C03596=1036.829,292.266,-117.984,171.449,43.308,158.322
C03597=1036.819,291.919,-117.939,171.445,43.306,158.321
C03598=1036.810,291.572,-117.895,171.438,43.304,158.320
C03599=1036.801,291.226,-117.849,171.434,43.302,158.319
C03600=1036.791,290.879,-117.804,171.429,43.301,158.318
C03601=1036.784,290.631,-117.772,171.425,43.299,158.318
C03602=1036.777,290.384,-117.740,171.420,43.298,158.317
C03603=1036.771,290.136,-117.708,171.417,43.297,158.317
C03604=1036.763,289.888,-117.676,171.413,43.296,158.316
C03605=1036.757,289.640,-117.644,171.409,43.295,158.316
C03606=1036.750,289.393,-117.612,171.406,43.294,158.315
C03607=1036.744,289.144,-117.580,171.402,43.292,158.314
C03608=1036.737,288.896,-117.549,171.398,43.291,158.314
C03609=1036.729,288.648,-117.516,171.395,43.290,158.313
C03610=1036.723,288.401,-117.485,171.391,43.288,158.313
C03611=1036.716,288.153,-117.453,171.386,43.287,158.312
C03612=1036.710,287.905,-117.420,171.383,43.286,158.311
C03613=1036.703,287.657,-117.389,171.379,43.285,158.311
C03614=1036.696,287.410,-117.357,171.375,43.284,158.310
C03615=1036.689,287.162,-117.325,171.372,43.283,158.310
C03616=1036.682,286.913,-117.294,171.368,43.281,158.309
C03617=1036.675,286.666,-117.261,171.364,43.280,158.309
C03618=1036.669,286.418,-117.230,171.361,43.279,158.308
C03619=1036.662,286.170,-117.198,171.357,43.278,158.308
C03620=1036.655,285.922,-117.167,171.354,43.277,158.307
C03621=1036.648,285.675,-117.134,171.350,43.276,158.307
C03622=1036.642,285.427,-117.103,171.346,43.275,158.306
C03623=1036.634,285.178,-117.071,171.343,43.274,158.306
C03624=1036.627,284.930,-117.040,171.339,43.272,158.305
C03625=1036.621,284.683,-117.008,171.336,43.272,158.305
C03626=1036.613,284.435,-116.978,171.331,43.270,158.304
C03627=1036.607,284.187,-116.946,171.327,43.269,158.303
C03628=1036.600,283.940,-116.914,171.323,43.268,158.303
C03629=1036.593,283.692,-116.883,171.320,43.267,158.302
C03630=1036.586,283.444,-116.851,171.316,43.266,158.302
C03631=1036.579,283.196,-116.820,171.313,43.265,158.301
C03632=1036.573,282.948,-116.788,171.309,43.264,158.301
C03633=1036.566,282.700,-116.757,171.305,43.263,158.300
C03634=1036.559,282.452,-116.725,171.302,43.261,158.300
C03635=1036.552,282.204,-116.694,171.298,43.261,158.299
C03636=1036.546,281.957,-116.663,171.295,43.259,158.299
C03637=1036.539,281.709,-116.631,171.291,43.258,158.298
C03638=1036.532,281.461,-116.600,171.287,43.257,158.298
C03639=1036.526,281.213,-116.568,171.284,43.256,158.297
C03640=1036.519,280.965,-116.537,171.280,43.255,158.297
C03641=1036.512,280.717,-116.505,171.277,43.254,158.296
C03642=1036.506,280.468,-116.475,171.273,43.253,158.295
C03643=1036.499,280.221,-116.443,171.270,43.252,158.295
C03644=1036.492,279.973,-116.412,171.266,43.251,158.294
C03645=1036.485,279.725,-116.380,171.262,43.250,158.294
C03646=1036.479,279.477,-116.349,171.259,43.249,158.293
C03647=1036.472,279.229,-116.317,171.255,43.247,158.293
C03648=1036.465,278.981,-116.286,171.252,43.247,158.292
C03649=1036.459,278.733,-116.255,171.249,43.245,158.292
C03650=1036.452,278.485,-116.224,171.245,43.244,158.291
C03651=1036.445,278.237,-116.193,171.242,43.243,158.291
C03652=1036.438,277.989,-116.162,171.238,43.242,158.290
C03653=1036.429,277.655,-116.119,171.233,43.241,158.290
C03654=1036.420,277.319,-116.078,171.229,43.240,158.289
C03655=1036.411,276.985,-116.036,171.224,43.238,158.288
C03656=1036.401,276.651,-115.994,171.219,43.237,158.288
C03657=1036.395,276.402,-115.964,171.216,43.236,158.287
C03658=1036.388,276.154,-115.932,171.212,43.235,158.287
C03659=1036.382,275.906,-115.902,171.208,43.234,158.286
C03660=1036.374,275.658,-115.871,171.205,43.233,158.286
C03661=1036.368,275.411,-115.840,171.201,43.232,158.285
C03662=1036.362,275.162,-115.809,171.198,43.231,158.285
C03663=1036.354,274.915,-115.778,171.194,43.230,158.284
C03664=1036.348,274.666,-115.747,171.191,43.229,158.284
C03665=1036.341,274.418,-115.716,171.187,43.228,158.283
C03666=1036.335,274.170,-115.685,171.185,43.227,158.283
C03667=1036.328,273.923,-115.655,171.181,43.226,158.282
C03668=1036.321,273.674,-115.624,171.177,43.225,158.282
C03669=1036.314,273.427,-115.593,171.174,43.224,158.281
C03670=1036.308,273.178,-115.562,171.170,43.223,158.281
C03671=1036.301,272.930,-115.531,171.167,43.222,158.280
C03672=1036.294,272.682,-115.501,171.163,43.222,158.280
C03673=1036.288,272.434,-115.471,171.160,43.220,158.279
C03674=1036.280,272.187,-115.440,171.156,43.220,158.279
C03675=1036.274,271.938,-115.409,171.153,43.219,158.279
C03676=1036.267,271.690,-115.378,171.150,43.217,158.278
C03677=1036.260,271.442,-115.347,171.147,43.217,158.278
C03678=1036.254,271.194,-115.317,171.143,43.216,158.277
C03679=1036.247,270.947,-115.286,171.139,43.215,158.277
C03680=1036.240,270.698,-115.256,171.136,43.214,158.276
C03681=1036.233,270.450,-115.225,171.132,43.213,158.276
C03682=1036.227,270.202,-115.195,171.129,43.212,158.275
C03683=1036.220,269.955,-115.164,171.126,43.211,158.275
C03684=1036.214,269.706,-115.134,171.123,43.210,158.274
C03685=1036.206,269.458,-115.103,171.119,43.210,158.274
C03686=1036.201,269.210,-115.073,171.116,43.208,158.273
C03687=1036.193,268.962,-115.042,171.112,43.208,158.273
C03688=1036.187,268.714,-115.011,171.109,43.207,158.272
C03689=1036.180,268.466,-114.981,171.105,43.206,158.272
C03690=1036.173,268.218,-114.952,171.103,43.205,158.272
C03691=1036.167,267.970,-114.921,171.099,43.204,158.271
C03692=1036.159,267.721,-114.891,171.096,43.203,158.271
C03693=1036.154,267.474,-114.860,171.092,43.203,158.270
C03694=1036.146,267.225,-114.830,171.089,43.202,158.270
C03695=1036.140,266.977,-114.799,171.085,43.201,158.269
C03696=1036.133,266.730,-114.769,171.083,43.200,158.269
C03697=1036.126,266.482,-114.739,171.079,43.199,158.268
C03698=1036.120,266.233,-114.708,171.076,43.198,158.268
C03699=1036.113,265.986,-114.679,171.072,43.198,158.268
C03700=1036.106,265.737,-114.648,171.069,43.197,158.267
C03701=1036.099,265.489,-114.618,171.066,43.195,158.267
C03702=1036.093,265.241,-114.588,171.063,43.195,158.266
C03703=1036.086,264.993,-114.559,171.059,43.194,158.266
C03704=1036.079,264.744,-114.528,171.056,43.193,158.265
C03705=1036.073,264.497,-114.498,171.052,43.193,158.265
C03706=1036.066,264.248,-114.468,171.050,43.192,158.265
C03707=1036.059,264.000,-114.438,171.046,43.191,158.264
C03708=1036.052,263.753,-114.408,171.043,43.190,158.264
C03709=1036.044,263.422,-114.368,171.038,43.189,158.263
C03710=1036.035,263.092,-114.328,171.035,43.188,158.263
C03711=1036.026,262.762,-114.287,171.030,43.187,158.262
C03712=1036.017,262.432,-114.248,171.025,43.185,158.261
C03713=1036.009,262.184,-114.218,171.022,43.185,158.261
C03714=1036.004,261.935,-114.188,171.019,43.184,158.260
C03715=1035.997,261.687,-114.158,171.016,43.183,158.260
C03716=1035.990,261.440,-114.128,171.012,43.182,158.260
C03717=1035.983,261.192,-114.098,171.009,43.182,158.259
C03718=1035.976,260.943,-114.069,171.006,43.181,158.259
C03719=1035.970,260.695,-114.039,171.003,43.180,158.258
C03720=1035.963,260.446,-114.009,171.000,43.179,158.258
C03721=1035.956,260.199,-113.980,170.996,43.179,158.258
C03722=1035.948,259.951,-113.950,170.993,43.179,158.257
C03723=1035.942,259.702,-113.921,170.990,43.178,158.257
C03724=1035.935,259.455,-113.891,170.987,43.177,158.256
C03725=1035.928,259.206,-113.862,170.983,43.176,158.256
C03726=1035.922,258.958,-113.832,170.980,43.176,158.256
C03727=1035.915,258.709,-113.802,170.978,43.175,158.255
C03728=1035.908,258.462,-113.773,170.974,43.174,158.255
C03729=1035.901,258.214,-113.743,170.971,43.173,158.254
C03730=1035.894,257.965,-113.713,170.967,43.173,158.254
C03731=1035.887,257.718,-113.684,170.965,43.172,158.254
C03732=1035.880,257.469,-113.655,170.961,43.172,158.253
C03733=1035.874,257.221,-113.626,170.958,43.171,158.253
C03734=1035.867,256.972,-113.595,170.955,43.170,158.252
C03735=1035.860,256.724,-113.566,170.952,43.169,158.252
C03736=1035.853,256.476,-113.536,170.949,43.169,158.252
C03737=1035.847,256.228,-113.507,170.945,43.168,158.251
C03738=1035.840,255.980,-113.477,170.943,43.167,158.251
C03739=1035.833,255.732,-113.449,170.939,43.167,158.251
C03740=1035.826,255.483,-113.419,170.936,43.166,158.250
C03741=1035.819,255.236,-113.389,170.933,43.165,158.250
C03742=1035.813,254.987,-113.360,170.930,43.165,158.249
C03743=1035.806,254.739,-113.330,170.927,43.164,158.249
C03744=1035.800,254.491,-113.301,170.923,43.163,158.248
C03745=1035.793,254.242,-113.272,170.921,43.162,158.248
C03746=1035.786,253.995,-113.243,170.917,43.162,158.248
C03747=1035.779,253.746,-113.213,170.914,43.161,158.247
C03748=1035.772,253.498,-113.184,170.912,43.161,158.247
C03749=1035.765,253.250,-113.154,170.908,43.160,158.247
C03750=1035.759,253.002,-113.125,170.905,43.159,158.246
C03751=1035.753,252.754,-113.096,170.902,43.158,158.246
C03752=1035.746,252.505,-113.067,170.899,43.158,158.245
C03753=1035.739,252.258,-113.037,170.895,43.157,158.245
C03754=1035.732,252.009,-113.008,170.893,43.157,158.245
C03755=1035.726,251.761,-112.979,170.890,43.156,158.244
C03756=1035.719,251.513,-112.950,170.886,43.155,158.244
C03757=1035.712,251.264,-112.921,170.884,43.154,158.244
C03758=1035.706,251.016,-112.891,170.880,43.154,158.243
C03759=1035.700,250.768,-112.862,170.877,43.153,158.243
C03760=1035.692,250.520,-112.833,170.874,43.153,158.242
C03761=1035.686,250.271,-112.804,170.871,43.152,158.242
C03762=1035.680,250.023,-112.775,170.869,43.151,158.242
C03763=1035.673,249.774,-112.745,170.865,43.150,158.241
C03764=1035.666,249.527,-112.716,170.862,43.149,158.241
C03765=1035.657,249.195,-112.677,170.858,43.149,158.240
C03766=1035.648,248.864,-112.638,170.854,43.148,158.240
C03767=1035.640,248.532,-112.600,170.850,43.147,158.239
C03768=1035.631,248.201,-112.560,170.846,43.146,158.239
C03769=1035.625,247.953,-112.531,170.843,43.145,158.238
C03770=1035.618,247.705,-112.502,170.840,43.145,158.238
C03771=1035.611,247.456,-112.473,170.837,43.144,158.238
C03772=1035.604,247.208,-112.444,170.834,43.144,158.237
C03773=1035.598,246.960,-112.415,170.831,43.143,158.237
C03774=1035.592,246.712,-112.386,170.828,43.142,158.237
C03775=1035.585,246.463,-112.357,170.825,43.141,158.236
C03776=1035.579,246.215,-112.328,170.822,43.140,158.236
C03777=1035.572,245.967,-112.299,170.819,43.140,158.236
C03778=1035.566,245.719,-112.270,170.816,43.139,158.235
C03779=1035.559,245.470,-112.241,170.813,43.139,158.235
C03780=1035.553,245.222,-112.212,170.811,43.138,158.234
C03781=1035.546,244.974,-112.183,170.807,43.137,158.234
C03782=1035.539,244.726,-112.154,170.805,43.137,158.234
C03783=1035.533,244.477,-112.126,170.801,43.136,158.233
C03784=1035.527,244.228,-112.097,170.798,43.135,158.233
C03785=1035.520,243.980,-112.068,170.796,43.135,158.233
C03786=1035.513,243.732,-112.039,170.792,43.134,158.232
C03787=1035.506,243.484,-112.011,170.790,43.134,158.232
C03788=1035.500,243.235,-111.982,170.786,43.133,158.232
C03789=1035.493,242.987,-111.954,170.784,43.133,158.231
C03790=1035.487,242.739,-111.925,170.781,43.132,158.231
C03791=1035.480,242.491,-111.896,170.778,43.132,158.230
C03792=1035.474,242.243,-111.868,170.775,43.131,158.230
C03793=1035.467,241.994,-111.838,170.771,43.130,158.230
C03794=1035.460,241.746,-111.810,170.769,43.130,158.229
C03795=1035.453,241.498,-111.781,170.766,43.129,158.229
C03796=1035.447,241.249,-111.753,170.763,43.128,158.229
C03797=1035.441,241.001,-111.724,170.760,43.128,158.228
C03798=1035.434,240.753,-111.696,170.758,43.127,158.228
C03799=1035.428,240.505,-111.667,170.754,43.126,158.228
C03800=1035.420,240.256,-111.639,170.752,43.126,158.227
C03801=1035.413,240.008,-111.610,170.748,43.125,158.227
C03802=1035.407,239.759,-111.582,170.746,43.125,158.227
C03803=1035.400,239.512,-111.553,170.743,43.124,158.226
C03804=1035.393,239.263,-111.526,170.740,43.124,158.226
C03805=1035.387,239.014,-111.496,170.737,43.123,158.226
C03806=1035.380,238.766,-111.468,170.735,43.123,158.225
C03807=1035.373,238.518,-111.440,170.731,43.122,158.225
C03808=1035.366,238.270,-111.412,170.729,43.122,158.225
C03809=1035.360,238.022,-111.383,170.726,43.121,158.224
C03810=1035.353,237.773,-111.356,170.723,43.121,158.224
C03811=1035.346,237.525,-111.327,170.720,43.120,158.224
C03812=1035.340,237.277,-111.299,170.718,43.120,158.223
C03813=1035.333,237.028,-111.270,170.714,43.119,158.223
C03814=1035.326,236.780,-111.242,170.712,43.119,158.223
C03815=1035.319,236.531,-111.214,170.709,43.118,158.222
C03816=1035.312,236.283,-111.186,170.706,43.118,158.222
C03817=1035.306,236.035,-111.158,170.703,43.117,158.222
C03818=1035.300,235.787,-111.129,170.700,43.117,158.221
C03819=1035.293,235.538,-111.102,170.697,43.116,158.221
C03820=1035.286,235.290,-111.074,170.695,43.116,158.221
C03821=1035.277,234.952,-111.035,170.690,43.115,158.220
C03822=1035.269,234.615,-110.997,170.687,43.114,158.220
C03823=1035.259,234.278,-110.958,170.682,43.114,158.219
C03824=1035.250,233.940,-110.920,170.679,43.113,158.219
C03825=1035.243,233.691,-110.892,170.677,43.113,158.219
C03826=1035.236,233.444,-110.864,170.673,43.112,158.218
C03827=1035.230,233.195,-110.836,170.671,43.112,158.218
C03828=1035.223,232.947,-110.808,170.667,43.111,158.218
C03829=1035.217,232.698,-110.780,170.665,43.111,158.217
C03830=1035.210,232.450,-110.752,170.662,43.110,158.217
C03831=1035.203,232.202,-110.724,170.660,43.110,158.217
C03832=1035.197,231.953,-110.696,170.657,43.109,158.216
C03833=1035.191,231.704,-110.668,170.654,43.109,158.216
C03834=1035.184,231.457,-110.639,170.651,43.108,158.216
C03835=1035.177,231.208,-110.612,170.648,43.108,158.215
C03836=1035.170,230.960,-110.584,170.646,43.107,158.215
C03837=1035.164,230.711,-110.556,170.642,43.107,158.215
C03838=1035.157,230.463,-110.528,170.640,43.106,158.214
C03839=1035.150,230.214,-110.501,170.638,43.106,158.214
C03840=1035.144,229.966,-110.473,170.635,43.105,158.214
C03841=1035.137,229.718,-110.445,170.632,43.105,158.213
C03842=1035.130,229.470,-110.417,170.629,43.104,158.213
C03843=1035.123,229.221,-110.389,170.627,43.104,158.213
C03844=1035.117,228.974,-110.362,170.624,43.103,158.213
C03845=1035.110,228.725,-110.334,170.621,43.103,158.212
C03846=1035.104,228.477,-110.306,170.618,43.102,158.212
C03847=1035.097,228.228,-110.279,170.615,43.102,158.212
C03848=1035.090,227.980,-110.251,170.613,43.101,158.211
C03849=1035.084,227.731,-110.223,170.609,43.101,158.211
C03850=1035.077,227.483,-110.195,170.607,43.101,158.211
C03851=1035.070,227.234,-110.168,170.605,43.101,158.211
C03852=1035.064,226.986,-110.140,170.602,43.100,158.210
C03853=1035.057,226.738,-110.112,170.599,43.100,158.210
C03854=1035.050,226.489,-110.085,170.596,43.099,158.210
C03855=1035.043,226.241,-110.057,170.594,43.099,158.209
C03856=1035.037,225.992,-110.030,170.591,43.098,158.209
C03857=1035.030,225.743,-110.003,170.588,43.098,158.209
C03858=1035.023,225.495,-109.975,170.586,43.097,158.208
C03859=1035.017,225.247,-109.947,170.582,43.097,158.208
C03860=1035.009,224.998,-109.920,170.580,43.097,158.208
C03861=1035.003,224.751,-109.893,170.578,43.096,158.207
C03862=1034.996,224.502,-109.865,170.575,43.096,158.207
C03863=1034.990,224.253,-109.838,170.572,43.096,158.207
C03864=1034.983,224.005,-109.810,170.570,43.095,158.207
C03865=1034.977,223.756,-109.782,170.567,43.095,158.206
C03866=1034.969,223.508,-109.755,170.564,43.094,158.206
C03867=1034.963,223.260,-109.728,170.561,43.094,158.206
C03868=1034.956,223.011,-109.701,170.559,43.093,158.205
C03869=1034.950,222.763,-109.673,170.556,43.093,158.205
C03870=1034.943,222.515,-109.645,170.553,43.093,158.205
C03871=1034.936,222.266,-109.618,170.551,43.092,158.205
C03872=1034.930,222.017,-109.591,170.549,43.092,158.204
C03873=1034.923,221.769,-109.564,170.545,43.092,158.204
C03874=1034.916,221.520,-109.536,170.543,43.091,158.204
C03875=1034.910,221.273,-109.508,170.541,43.090,158.203
C03876=1034.903,221.024,-109.482,170.537,43.090,158.203
C03877=1034.894,220.679,-109.444,170.534,43.090,158.203
C03878=1034.885,220.334,-109.406,170.530,43.089,158.202
C03879=1034.875,219.989,-109.368,170.527,43.088,158.202
C03880=1034.866,219.644,-109.330,170.523,43.087,158.201
C03881=1034.860,219.395,-109.302,170.520,43.087,158.201
C03882=1034.853,219.148,-109.276,170.518,43.087,158.201
C03883=1034.846,218.899,-109.249,170.516,43.087,158.201
C03884=1034.839,218.651,-109.221,170.513,43.087,158.200
C03885=1034.833,218.402,-109.194,170.510,43.086,158.200
C03886=1034.825,218.154,-109.167,170.508,43.085,158.200
C03887=1034.819,217.905,-109.140,170.505,43.085,158.200
C03888=1034.812,217.657,-109.113,170.502,43.085,158.199
C03889=1034.806,217.408,-109.086,170.500,43.085,158.199
C03890=1034.798,217.160,-109.059,170.497,43.084,158.199
C03891=1034.792,216.911,-109.032,170.494,43.084,158.198
C03892=1034.786,216.663,-109.005,170.492,43.083,158.198
C03893=1034.779,216.414,-108.979,170.489,43.083,158.198
C03894=1034.772,216.166,-108.951,170.487,43.083,158.198
C03895=1034.765,215.917,-108.924,170.484,43.082,158.197
C03896=1034.759,215.669,-108.897,170.481,43.082,158.197
C03897=1034.752,215.421,-108.871,170.479,43.082,158.197
C03898=1034.745,215.172,-108.844,170.477,43.081,158.197
C03899=1034.738,214.924,-108.816,170.474,43.081,158.196
C03900=1034.732,214.675,-108.790,170.471,43.080,158.196
C03901=1034.725,214.427,-108.763,170.469,43.080,158.196
C03902=1034.718,214.178,-108.736,170.466,43.080,158.196
C03903=1034.711,213.929,-108.709,170.464,43.079,158.195
C03904=1034.705,213.681,-108.682,170.461,43.079,158.195
C03905=1034.698,213.433,-108.655,170.459,43.079,158.195
C03906=1034.692,213.184,-108.628,170.456,43.078,158.194
C03907=1034.685,212.936,-108.602,170.454,43.078,158.194
C03908=1034.678,212.687,-108.575,170.451,43.078,158.194
C03909=1034.671,212.438,-108.548,170.449,43.078,158.194
C03910=1034.665,212.191,-108.521,170.446,43.077,158.193
C03911=1034.658,211.942,-108.494,170.444,43.076,158.193
C03912=1034.652,211.693,-108.467,170.441,43.076,158.193
C03913=1034.645,211.445,-108.441,170.438,43.076,158.193
C03914=1034.639,211.196,-108.414,170.436,43.076,158.192
C03915=1034.631,210.948,-108.387,170.434,43.075,158.192
C03916=1034.625,210.700,-108.361,170.430,43.075,158.192
C03917=1034.618,210.451,-108.333,170.428,43.074,158.191
C03918=1034.611,210.202,-108.307,170.426,43.074,158.191
C03919=1034.605,209.954,-108.281,170.424,43.074,158.191
C03920=1034.598,209.705,-108.254,170.420,43.074,158.191
C03921=1034.591,209.457,-108.228,170.418,43.073,158.190
C03922=1034.585,209.208,-108.201,170.416,43.073,158.190
C03923=1034.578,208.960,-108.174,170.414,43.073,158.190
C03924=1034.571,208.712,-108.148,170.411,43.072,158.190
C03925=1034.564,208.463,-108.121,170.408,43.072,158.189
C03926=1034.558,208.214,-108.094,170.406,43.071,158.189
C03927=1034.551,207.966,-108.068,170.404,43.071,158.189
C03928=1034.544,207.717,-108.042,170.401,43.071,158.189
C03929=1034.537,207.469,-108.015,170.398,43.071,158.188
C03930=1034.531,207.220,-107.989,170.396,43.071,158.188
C03931=1034.524,206.972,-107.962,170.394,43.070,158.188
C03932=1034.518,206.723,-107.936,170.391,43.070,158.188
C03933=1034.508,206.384,-107.900,170.388,43.069,158.187
C03934=1034.498,206.045,-107.864,170.385,43.069,158.187
C03935=1034.490,205.706,-107.828,170.381,43.068,158.187
C03936=1034.481,205.366,-107.792,170.378,43.068,158.186
C03937=1034.454,204.316,-107.686,170.052,42.963,158.140
C03938=1034.448,204.068,-107.661,170.048,42.964,158.140
C03939=1034.443,203.820,-107.636,170.045,42.965,158.140
C03940=1034.436,203.571,-107.611,170.042,42.965,158.140
C03941=1034.430,203.322,-107.586,170.038,42.966,158.139
C03942=1034.424,203.073,-107.561,170.034,42.966,158.139
C03943=1034.417,202.825,-107.536,170.031,42.966,158.139
C03944=1034.412,202.577,-107.511,170.027,42.967,158.139
C03945=1034.406,202.327,-107.486,170.024,42.967,158.139
C03946=1034.400,202.079,-107.461,170.021,42.968,158.139
C03947=1034.393,201.830,-107.435,170.018,42.968,158.138
C03948=1034.388,201.581,-107.411,170.014,42.969,158.138
C03949=1034.381,201.333,-107.386,170.011,42.969,158.138
C03950=1034.375,201.084,-107.361,170.008,42.970,158.138
C03951=1034.369,200.835,-107.337,170.004,42.970,158.138
C03952=1034.363,200.587,-107.311,170.001,42.971,158.138
C03953=1034.357,200.337,-107.287,169.998,42.971,158.137
C03954=1034.351,200.090,-107.262,169.994,42.972,158.137
C03955=1034.345,199.840,-107.238,169.991,42.972,158.137
C03956=1034.338,199.592,-107.213,169.987,42.973,158.137
C03957=1034.332,199.343,-107.188,169.984,42.973,158.137
C03958=1034.325,199.094,-107.163,169.980,42.974,158.137
C03959=1034.320,198.846,-107.139,169.977,42.975,158.137
C03960=1034.313,198.597,-107.114,169.974,42.975,158.137
C03961=1034.307,198.348,-107.090,169.970,42.976,158.136
C03962=1034.300,198.099,-107.066,169.967,42.977,158.136
C03963=1034.295,197.851,-107.041,169.964,42.978,158.136
C03964=1034.288,197.602,-107.017,169.960,42.978,158.136
C03965=1034.282,197.353,-106.991,169.957,42.979,158.136
C03966=1034.275,197.104,-106.967,169.954,42.979,158.136
C03967=1034.270,196.856,-106.943,169.951,42.980,158.136
C03968=1034.263,196.608,-106.918,169.947,42.980,158.136
C03969=1034.257,196.358,-106.894,169.944,42.981,158.135
C03970=1034.252,196.110,-106.870,169.941,42.981,158.135
C03971=1034.245,195.861,-106.845,169.937,42.982,158.135
C03972=1034.239,195.612,-106.820,169.934,42.983,158.135
C03973=1034.233,195.364,-106.797,169.931,42.984,158.135
C03974=1034.227,195.115,-106.771,169.928,42.984,158.135
C03975=1034.220,194.866,-106.747,169.924,42.985,158.135
C03976=1034.215,194.617,-106.723,169.921,42.985,158.135
C03977=1034.208,194.369,-106.699,169.918,42.986,158.135
C03978=1034.202,194.120,-106.674,169.915,42.986,158.134
C03979=1034.196,193.872,-106.650,169.912,42.987,158.134
C03980=1034.190,193.622,-106.625,169.908,42.988,158.134
C03981=1034.183,193.373,-106.601,169.905,42.989,158.134
C03982=1034.178,193.125,-106.577,169.902,42.989,158.134
C03983=1034.171,192.876,-106.552,169.899,42.990,158.134
C03984=1034.166,192.628,-106.528,169.895,42.991,158.134
C03985=1034.159,192.379,-106.504,169.892,42.991,158.134
C03986=1034.153,192.129,-106.479,169.889,42.992,158.133
C03987=1034.147,191.881,-106.456,169.886,42.993,158.133
C03988=1034.141,191.632,-106.431,169.883,42.993,158.133
C03989=1034.135,191.384,-106.407,169.879,42.994,158.133
C03990=1034.128,191.135,-106.383,169.876,42.994,158.133
C03991=1034.122,190.886,-106.358,169.873,42.995,158.133
C03992=1034.116,190.638,-106.334,169.870,42.995,158.133
C03993=1034.110,190.388,-106.310,169.867,42.997,158.133
C03994=1034.104,190.140,-106.286,169.864,42.997,158.133
C03995=1034.098,189.891,-106.261,169.860,42.998,158.133
C03996=1034.092,189.643,-106.238,169.857,42.998,158.132
C03997=1034.086,189.393,-106.213,169.854,42.999,158.132
C03998=1034.080,189.110,-106.185,169.850,43.000,158.132
C03999=1034.073,188.826,-106.158,169.847,43.001,158.132
C04000=1034.066,188.541,-106.130,169.843,43.001,158.132
C04001=1034.059,188.258,-106.103,169.840,43.002,158.132
C04002=1034.053,188.010,-106.079,169.837,43.002,158.132
C04003=1034.047,187.760,-106.054,169.833,43.004,158.132
C04004=1034.041,187.512,-106.031,169.830,43.004,158.132
C04005=1034.035,187.263,-106.006,169.827,43.005,158.131
C04006=1034.029,187.015,-105.982,169.824,43.005,158.131
C04007=1034.023,186.766,-105.958,169.821,43.006,158.131
C04008=1034.017,186.517,-105.934,169.818,43.007,158.131
C04009=1034.011,186.267,-105.911,169.815,43.007,158.131
C04010=1034.006,186.019,-105.887,169.812,43.008,158.131
C04011=1034.000,185.770,-105.863,169.808,43.009,158.131
C04012=1033.994,185.521,-105.838,169.805,43.010,158.131
C04013=1033.988,185.273,-105.815,169.802,43.010,158.131
C04014=1033.982,185.024,-105.790,169.799,43.011,158.131
C04015=1033.976,184.775,-105.766,169.796,43.011,158.130
C04016=1033.970,184.527,-105.742,169.793,43.012,158.130
C04017=1033.964,184.277,-105.719,169.790,43.013,158.130
C04018=1033.958,184.029,-105.695,169.787,43.013,158.130
C04019=1033.952,183.780,-105.671,169.784,43.014,158.130
C04020=1033.946,183.531,-105.647,169.781,43.015,158.130
C04021=1033.941,183.283,-105.623,169.778,43.016,158.130
C04022=1033.935,183.033,-105.599,169.774,43.016,158.130
C04023=1033.928,182.785,-105.576,169.771,43.017,158.130
C04024=1033.922,182.536,-105.552,169.768,43.018,158.130
C04025=1033.915,182.287,-105.529,169.765,43.019,158.130
C04026=1033.909,182.038,-105.505,169.762,43.020,158.130
C04027=1033.903,181.789,-105.482,169.759,43.021,158.130
C04028=1033.897,181.541,-105.459,169.756,43.022,158.130
C04029=1033.891,181.292,-105.435,169.752,43.023,158.129
C04030=1033.885,181.043,-105.412,169.750,43.024,158.129
C04031=1033.878,180.794,-105.388,169.747,43.024,158.129
C04032=1033.872,180.545,-105.365,169.744,43.025,158.129
C04033=1033.865,180.296,-105.342,169.741,43.026,158.129
C04034=1033.859,180.048,-105.318,169.738,43.027,158.129
C04035=1033.853,179.799,-105.295,169.735,43.028,158.129
C04036=1033.847,179.550,-105.271,169.731,43.029,158.129
C04037=1033.841,179.301,-105.248,169.728,43.030,158.129
C04038=1033.834,179.052,-105.224,169.725,43.031,158.129
C04039=1033.828,178.803,-105.202,169.722,43.032,158.129
C04040=1033.822,178.555,-105.178,169.719,43.033,158.129
C04041=1033.816,178.306,-105.155,169.716,43.033,158.129
C04042=1033.810,178.057,-105.131,169.714,43.035,158.129
C04043=1033.804,177.808,-105.108,169.711,43.035,158.129
C04044=1033.797,177.559,-105.085,169.708,43.036,158.129
C04045=1033.791,177.311,-105.061,169.704,43.038,158.129
C04046=1033.785,177.062,-105.039,169.701,43.038,158.129
C04047=1033.778,176.813,-105.015,169.698,43.039,158.129
C04048=1033.773,176.564,-104.992,169.695,43.040,158.129
C04049=1033.767,176.315,-104.969,169.692,43.041,158.129
C04050=1033.760,176.066,-104.945,169.689,43.042,158.129
C04051=1033.754,175.817,-104.922,169.686,43.043,158.128
C04052=1033.748,175.569,-104.900,169.683,43.044,158.129
C04053=1033.742,175.320,-104.876,169.680,43.044,158.128
C04054=1033.736,175.071,-104.853,169.678,43.045,158.128
C04055=1033.730,174.822,-104.830,169.675,43.047,158.128
C04056=1033.724,174.573,-104.807,169.672,43.047,158.128
C04057=1033.717,174.324,-104.784,169.669,43.048,158.128
C04058=1033.711,174.076,-104.761,169.666,43.049,158.128
C04059=1033.705,173.827,-104.738,169.663,43.050,158.128
C04060=1033.699,173.578,-104.714,169.660,43.051,158.128
C04061=1033.694,173.329,-104.691,169.656,43.052,158.128
C04062=1033.687,173.068,-104.667,169.653,43.053,158.128
C04063=1033.680,172.806,-104.643,169.650,43.054,158.128
C04064=1033.673,172.545,-104.618,169.647,43.055,158.128
C04065=1033.668,172.284,-104.594,169.645,43.056,158.128
C04066=1033.662,172.035,-104.572,169.642,43.057,158.128
C04067=1033.655,171.786,-104.549,169.639,43.057,158.128
C04068=1033.649,171.537,-104.525,169.636,43.059,158.128
C04069=1033.644,171.288,-104.502,169.633,43.060,158.128
C04070=1033.638,171.040,-104.479,169.630,43.060,158.128
C04071=1033.631,170.791,-104.457,169.627,43.061,158.128
C04072=1033.625,170.541,-104.433,169.624,43.063,158.128
C04073=1033.619,170.292,-104.410,169.621,43.063,158.128
C04074=1033.614,170.044,-104.387,169.618,43.064,158.128
C04075=1033.608,169.795,-104.364,169.615,43.065,158.128
C04076=1033.601,169.547,-104.341,169.613,43.066,158.128
C04077=1033.595,169.298,-104.318,169.610,43.067,158.128
C04078=1033.590,169.049,-104.295,169.607,43.068,158.127
C04079=1033.583,168.799,-104.272,169.604,43.069,158.127
C04080=1033.578,168.550,-104.249,169.601,43.070,158.128
C04081=1033.571,168.302,-104.227,169.598,43.070,158.127
C04082=1033.565,168.053,-104.204,169.595,43.072,158.127
C04083=1033.560,167.804,-104.181,169.592,43.073,158.127
C04084=1033.554,167.555,-104.158,169.589,43.073,158.127
C04085=1033.547,167.307,-104.136,169.586,43.074,158.127
C04086=1033.542,167.058,-104.113,169.584,43.076,158.127
C04087=1033.536,166.809,-104.090,169.581,43.076,158.127
C04088=1033.530,166.560,-104.067,169.578,43.077,158.127
C04089=1033.525,166.311,-104.044,169.575,43.078,158.127
C04090=1033.517,166.062,-104.021,169.572,43.079,158.127
C04091=1033.512,165.813,-103.998,169.569,43.080,158.127
C04092=1033.506,165.564,-103.975,169.566,43.081,158.127
C04093=1033.500,165.315,-103.952,169.564,43.082,158.127
C04094=1033.494,165.066,-103.930,169.561,43.083,158.127
C04095=1033.488,164.818,-103.907,169.558,43.084,158.127
C04096=1033.482,164.569,-103.884,169.555,43.085,158.127
C04097=1033.477,164.320,-103.861,169.553,43.086,158.127
C04098=1033.470,164.071,-103.839,169.550,43.087,158.127
C04099=1033.464,163.822,-103.816,169.547,43.087,158.127
C04100=1033.459,163.573,-103.794,169.544,43.089,158.127
C04101=1033.453,163.324,-103.771,169.541,43.090,158.127
C04102=1033.447,163.052,-103.746,169.538,43.090,158.127
C04103=1033.441,162.780,-103.721,169.535,43.091,158.127
C04104=1033.434,162.509,-103.696,169.532,43.093,158.127
C04105=1033.427,162.237,-103.671,169.529,43.094,158.127
C04106=1033.422,161.987,-103.649,169.526,43.094,158.127
C04107=1033.416,161.738,-103.626,169.524,43.095,158.127
C04108=1033.410,161.489,-103.603,169.521,43.097,158.127
C04109=1033.404,161.241,-103.581,169.518,43.097,158.127
C04110=1033.398,160.993,-103.558,169.515,43.098,158.127
C04111=1033.393,160.743,-103.536,169.512,43.099,158.127
C04112=1033.387,160.494,-103.514,169.510,43.100,158.127
C04113=1033.381,160.246,-103.491,169.507,43.101,158.127
C04114=1033.375,159.997,-103.468,169.504,43.102,158.127
C04115=1033.370,159.747,-103.446,169.501,43.103,158.126
C04116=1033.363,159.499,-103.423,169.498,43.104,158.126
C04117=1033.357,159.250,-103.401,169.496,43.105,158.126
C04118=1033.351,159.000,-103.379,169.493,43.106,158.126
C04119=1033.345,158.752,-103.356,169.490,43.107,158.126
C04120=1033.339,158.503,-103.335,169.487,43.108,158.126
C04121=1033.333,158.254,-103.312,169.484,43.110,158.126
C04122=1033.327,158.005,-103.289,169.481,43.111,158.127
C04123=1033.320,157.756,-103.268,169.480,43.112,158.127
C04124=1033.315,157.507,-103.245,169.477,43.113,158.127
C04125=1033.308,157.258,-103.223,169.474,43.113,158.126
C04126=1033.302,156.973,-103.197,169.470,43.115,158.126
C04127=1033.295,156.688,-103.172,169.467,43.117,158.127
C04128=1033.288,156.404,-103.147,169.464,43.118,158.127
C04129=1033.281,156.118,-103.121,169.462,43.119,158.127
C04130=1033.274,155.869,-103.099,169.459,43.119,158.126
C04131=1033.269,155.621,-103.078,169.456,43.121,158.126
C04132=1033.262,155.372,-103.055,169.453,43.122,158.127
C04133=1033.257,155.123,-103.033,169.450,43.123,158.127
C04134=1033.251,154.874,-103.011,169.447,43.124,158.127
C04135=1033.244,154.625,-102.989,169.444,43.125,158.127
C04136=1033.239,154.376,-102.966,169.442,43.126,158.127
C04137=1033.232,154.127,-102.945,169.440,43.127,158.127
C04138=1033.226,153.878,-102.923,169.437,43.129,158.127
C04139=1033.220,153.629,-102.901,169.434,43.130,158.127
C04140=1033.214,153.380,-102.878,169.431,43.131,158.127
C04141=1033.209,153.132,-102.856,169.428,43.132,158.127
C04142=1033.202,152.883,-102.835,169.426,43.133,158.127
C04143=1033.196,152.633,-102.813,169.423,43.134,158.127
C04144=1033.190,152.385,-102.791,169.420,43.136,158.127
C04145=1033.184,152.136,-102.769,169.418,43.137,158.127
C04146=1033.178,151.886,-102.747,169.415,43.138,158.127
C04147=1033.172,151.637,-102.725,169.412,43.139,158.127
C04148=1033.166,151.389,-102.703,169.410,43.140,158.127
C04149=1033.160,151.140,-102.682,169.407,43.141,158.127
C04150=1033.154,150.891,-102.660,169.404,43.142,158.127
C04151=1033.147,150.642,-102.638,169.401,43.144,158.127
C04152=1033.142,150.392,-102.616,169.399,43.144,158.127
C04153=1033.136,150.143,-102.594,169.396,43.146,158.127
C04154=1033.130,149.895,-102.573,169.394,43.147,158.127
C04155=1033.124,149.646,-102.550,169.391,43.147,158.127
C04156=1033.118,149.397,-102.529,169.388,43.149,158.127
C04157=1033.111,149.148,-102.507,169.385,43.150,158.127
C04158=1033.105,148.899,-102.485,169.383,43.151,158.127
C04159=1033.099,148.651,-102.463,169.380,43.152,158.127
C04160=1033.093,148.401,-102.442,169.378,43.154,158.127
C04161=1033.088,148.152,-102.420,169.375,43.155,158.127
C04162=1033.082,147.903,-102.398,169.372,43.156,158.127
C04163=1033.075,147.654,-102.376,169.369,43.157,158.127
C04164=1033.070,147.405,-102.355,169.367,43.158,158.127
C04165=1033.064,147.156,-102.333,169.364,43.159,158.127
C04166=1033.057,146.907,-102.311,169.362,43.161,158.127
C04167=1033.051,146.658,-102.289,169.359,43.162,158.127
C04168=1033.045,146.409,-102.268,169.356,43.163,158.127
C04169=1033.039,146.160,-102.246,169.353,43.164,158.127
C04170=1033.033,145.911,-102.225,169.351,43.165,158.127
C04171=1033.027,145.662,-102.203,169.348,43.166,158.127
C04172=1033.020,145.413,-102.182,169.346,43.167,158.127
C04173=1033.015,145.165,-102.161,169.343,43.169,158.127
C04174=1033.008,144.915,-102.139,169.340,43.170,158.127
C04175=1033.002,144.666,-102.118,169.337,43.172,158.127
C04176=1032.996,144.417,-102.096,169.336,43.173,158.128
C04177=1032.991,144.168,-102.075,169.333,43.174,158.128
C04178=1032.984,143.919,-102.053,169.330,43.175,158.128
C04179=1032.978,143.670,-102.031,169.327,43.176,158.128
C04180=1032.972,143.421,-102.010,169.324,43.177,158.128
C04181=1032.966,143.173,-101.989,169.321,43.178,158.128
C04182=1032.960,142.923,-101.967,169.320,43.179,158.128
C04183=1032.953,142.674,-101.946,169.317,43.181,158.128
C04184=1032.947,142.425,-101.924,169.314,43.182,158.128
C04185=1032.942,142.176,-101.904,169.311,43.184,158.128
C04186=1032.936,141.927,-101.882,169.308,43.185,158.128
C04187=1032.930,141.677,-101.860,169.307,43.186,158.128
C04188=1032.924,141.429,-101.839,169.304,43.187,158.128
C04189=1032.917,141.180,-101.818,169.301,43.188,158.128
C04190=1032.911,140.895,-101.793,169.298,43.189,158.128
C04191=1032.904,140.610,-101.769,169.295,43.191,158.128
C04192=1032.897,140.325,-101.744,169.293,43.192,158.128
C04193=1032.890,140.040,-101.720,169.289,43.194,158.128
C04194=1032.884,139.791,-101.698,169.287,43.195,158.128
C04195=1032.878,139.542,-101.677,169.284,43.196,158.128
C04196=1032.872,139.292,-101.656,169.281,43.197,158.128
C04197=1032.866,139.043,-101.635,169.278,43.198,158.128
C04198=1032.860,138.795,-101.614,169.277,43.200,158.128
C04199=1032.854,138.546,-101.592,169.274,43.201,158.128
C04200=1032.848,138.296,-101.571,169.271,43.202,158.128
C04201=1032.842,138.047,-101.550,169.268,43.203,158.128
C04202=1032.835,137.798,-101.529,169.265,43.204,158.128
C04203=1032.829,137.549,-101.507,169.264,43.205,158.128
C04204=1032.824,137.300,-101.487,169.261,43.207,158.129
C04205=1032.817,137.051,-101.466,169.258,43.208,158.129
C04206=1032.811,136.802,-101.444,169.255,43.210,158.129
C04207=1032.805,136.553,-101.424,169.253,43.211,158.129
C04208=1032.799,136.304,-101.403,169.251,43.212,158.129
C04209=1032.793,136.055,-101.381,169.248,43.214,158.129
C04210=1032.787,135.806,-101.360,169.245,43.215,158.129
C04211=1032.780,135.557,-101.339,169.242,43.216,158.129
C04212=1032.775,135.308,-101.318,169.241,43.217,158.129
C04213=1032.769,135.058,-101.297,169.238,43.218,158.129
C04214=1032.763,134.810,-101.277,169.235,43.220,158.129
C04215=1032.756,134.561,-101.255,169.232,43.221,158.129
C04216=1032.750,134.311,-101.235,169.230,43.222,158.129
C04217=1032.744,134.063,-101.213,169.228,43.223,158.129
C04218=1032.738,133.813,-101.192,169.225,43.224,158.129
C04219=1032.732,133.565,-101.172,169.222,43.226,158.129
C04220=1032.726,133.315,-101.151,169.220,43.227,158.129
C04221=1032.719,133.066,-101.130,169.218,43.228,158.129
C04222=1032.714,132.818,-101.108,169.215,43.230,158.129
C04223=1032.708,132.568,-101.088,169.212,43.231,158.129
C04224=1032.702,132.320,-101.067,169.210,43.232,158.130
C04225=1032.696,132.070,-101.046,169.207,43.234,158.130
C04226=1032.689,131.822,-101.025,169.205,43.235,158.130
C04227=1032.684,131.572,-101.004,169.202,43.236,158.130
C04228=1032.678,131.323,-100.983,169.200,43.237,158.130
C04229=1032.671,131.074,-100.963,169.197,43.239,158.130
C04230=1032.666,130.825,-100.942,169.194,43.240,158.130
C04231=1032.659,130.576,-100.921,169.192,43.241,158.130
C04232=1032.653,130.327,-100.900,169.190,43.242,158.130
C04233=1032.647,130.078,-100.880,169.187,43.244,158.130
C04234=1032.641,129.828,-100.859,169.184,43.245,158.130
C04235=1032.634,129.580,-100.839,169.182,43.247,158.130
C04236=1032.628,129.330,-100.818,169.180,43.248,158.130
C04237=1032.622,129.081,-100.798,169.177,43.249,158.130
C04238=1032.615,128.833,-100.777,169.174,43.251,158.130
C04239=1032.610,128.583,-100.756,169.172,43.252,158.130
C04240=1032.604,128.334,-100.736,169.169,43.253,158.130
C04241=1032.597,128.086,-100.715,169.167,43.255,158.131
C04242=1032.591,127.836,-100.695,169.164,43.256,158.131
C04243=1032.585,127.586,-100.674,169.162,43.257,158.131
C04244=1032.579,127.338,-100.653,169.159,43.259,158.131
C04245=1032.572,127.089,-100.633,169.157,43.260,158.131
C04246=1032.567,126.840,-100.612,169.154,43.262,158.131
C04247=1032.560,126.590,-100.592,169.152,43.263,158.131
C04248=1032.554,126.342,-100.571,169.149,43.264,158.131
C04249=1032.547,126.092,-100.551,169.147,43.266,158.131
C04250=1032.542,125.843,-100.530,169.144,43.267,158.131
C04251=1032.535,125.594,-100.510,169.141,43.268,158.131
C04252=1032.529,125.345,-100.489,169.139,43.270,158.131
C04253=1032.523,125.097,-100.469,169.137,43.271,158.131
C04254=1032.516,124.811,-100.446,169.134,43.272,158.131
C04255=1032.509,124.526,-100.422,169.131,43.274,158.132
C04256=1032.502,124.241,-100.399,169.128,43.276,158.132
C04257=1032.495,123.954,-100.376,169.125,43.277,158.132
C04258=1032.489,123.706,-100.355,169.122,43.279,158.132
C04259=1032.482,123.457,-100.335,169.121,43.280,158.132
C04260=1032.476,123.208,-100.315,169.118,43.281,158.132
C04261=1032.471,122.959,-100.294,169.115,43.283,158.132
C04262=1032.465,122.709,-100.274,169.113,43.284,158.132
C04263=1032.459,122.461,-100.254,169.111,43.285,158.132
C04264=1032.452,122.212,-100.233,169.108,43.287,158.132
C04265=1032.446,121.963,-100.212,169.106,43.288,158.132
C04266=1032.440,121.713,-100.192,169.103,43.289,158.132
C04267=1032.434,121.464,-100.172,169.100,43.291,158.132
C04268=1032.428,121.215,-100.152,169.098,43.292,158.133
C04269=1032.422,120.966,-100.131,169.096,43.293,158.133
C04270=1032.416,120.717,-100.111,169.093,43.295,158.133
C04271=1032.410,120.468,-100.091,169.091,43.296,158.133
C04272=1032.403,120.218,-100.071,169.089,43.298,158.133
C04273=1032.398,119.969,-100.050,169.086,43.299,158.133
C04274=1032.392,119.720,-100.030,169.083,43.301,158.133
C04275=1032.385,119.472,-100.009,169.081,43.302,158.133
C04276=1032.379,119.223,-99.989,169.079,43.303,158.133
C04277=1032.373,118.973,-99.969,169.076,43.304,158.133
C04278=1032.367,118.724,-99.948,169.074,43.306,158.133
C04279=1032.361,118.475,-99.928,169.071,43.307,158.133
C04280=1032.355,118.226,-99.908,169.068,43.308,158.133
C04281=1032.349,117.977,-99.888,169.067,43.310,158.133
C04282=1032.344,117.728,-99.868,169.064,43.311,158.133
C04283=1032.337,117.478,-99.847,169.061,43.312,158.133
C04284=1032.331,117.230,-99.827,169.060,43.314,158.134
C04285=1032.325,116.981,-99.807,169.057,43.315,158.134
C04286=1032.319,116.731,-99.786,169.054,43.316,158.134
C04287=1032.313,116.482,-99.766,169.052,43.317,158.134
C04288=1032.307,116.233,-99.747,169.049,43.319,158.134
C04289=1032.301,115.984,-99.727,169.047,43.320,158.134
C04290=1032.295,115.734,-99.707,169.045,43.321,158.134
C04291=1032.290,115.485,-99.686,169.042,43.323,158.134
C04292=1032.284,115.236,-99.666,169.039,43.324,158.134
C04293=1032.277,114.987,-99.646,169.038,43.325,158.134
C04294=1032.271,114.738,-99.626,169.035,43.326,158.134
C04295=1032.265,114.489,-99.606,169.032,43.328,158.134
C04296=1032.260,114.240,-99.586,169.030,43.329,158.134
C04297=1032.253,113.991,-99.565,169.027,43.330,158.134
C04298=1032.247,113.742,-99.545,169.026,43.331,158.134
C04299=1032.241,113.493,-99.525,169.023,43.333,158.134
C04300=1032.236,113.243,-99.506,169.020,43.334,158.134
C04301=1032.230,112.994,-99.485,169.018,43.335,158.135
C04302=1032.224,112.745,-99.465,169.016,43.337,158.135
C04303=1032.218,112.496,-99.445,169.013,43.338,158.135
C04304=1032.211,112.247,-99.425,169.011,43.339,158.135
C04305=1032.205,111.997,-99.406,169.008,43.341,158.135
C04306=1032.199,111.749,-99.386,169.006,43.342,158.135
C04307=1032.193,111.500,-99.366,169.004,43.344,158.135
C04308=1032.186,111.250,-99.346,169.001,43.345,158.135
C04309=1032.180,111.001,-99.327,168.998,43.346,158.135
C04310=1032.174,110.752,-99.307,168.997,43.348,158.135
C04311=1032.168,110.503,-99.287,168.994,43.349,158.135
C04312=1032.162,110.253,-99.267,168.991,43.351,158.135
C04313=1032.156,110.004,-99.247,168.989,43.352,158.136
C04314=1032.150,109.755,-99.227,168.987,43.354,158.136
C04315=1032.144,109.506,-99.209,168.984,43.355,158.136
C04316=1032.137,109.257,-99.188,168.982,43.357,158.136
C04317=1032.131,109.008,-99.168,168.980,43.358,158.136
C04318=1032.124,108.723,-99.147,168.977,43.360,158.136
C04319=1032.117,108.437,-99.124,168.974,43.361,158.136
C04320=1032.110,108.151,-99.101,168.971,43.363,158.136
C04321=1032.103,107.866,-99.079,168.969,43.365,158.136
C04322=1032.097,107.617,-99.059,168.966,43.366,158.136
C04323=1032.090,107.368,-99.040,168.963,43.368,158.136
C04324=1032.084,107.119,-99.020,168.962,43.369,158.137
C04325=1032.079,106.869,-99.001,168.959,43.371,158.137
C04326=1032.073,106.621,-98.981,168.956,43.372,158.137
C04327=1032.066,106.371,-98.961,168.954,43.373,158.137
C04328=1032.060,106.122,-98.942,168.952,43.375,158.137
C04329=1032.054,105.873,-98.922,168.949,43.376,158.137
C04330=1032.048,105.624,-98.903,168.947,43.377,158.137
C04331=1032.042,105.375,-98.883,168.944,43.379,158.137
C04332=1032.035,105.126,-98.864,168.942,43.380,158.137
C04333=1032.029,104.876,-98.844,168.940,43.381,158.137
C04334=1032.023,104.627,-98.825,168.937,43.383,158.137
C04335=1032.017,104.378,-98.805,168.934,43.384,158.137
C04336=1032.011,104.129,-98.786,168.933,43.386,158.138
C04337=1032.005,103.880,-98.766,168.930,43.387,158.138
C04338=1031.999,103.631,-98.747,168.927,43.389,158.138
C04339=1031.992,103.381,-98.727,168.926,43.390,158.138
C04340=1031.986,103.132,-98.708,168.923,43.391,158.138
C04341=1031.980,102.883,-98.689,168.921,43.393,158.138
C04342=1031.974,102.634,-98.669,168.918,43.394,158.138
C04343=1031.969,102.384,-98.650,168.916,43.396,158.138
C04344=1031.962,102.136,-98.630,168.914,43.397,158.138
C04345=1031.956,101.886,-98.611,168.911,43.398,158.138
C04346=1031.950,101.638,-98.591,168.908,43.400,158.138
C04347=1031.944,101.389,-98.572,168.907,43.401,158.138
C04348=1031.938,101.138,-98.553,168.904,43.403,158.139
C04349=1031.932,100.890,-98.533,168.902,43.404,158.139
C04350=1031.926,100.640,-98.514,168.899,43.405,158.139
C04351=1031.919,100.391,-98.495,168.897,43.407,158.139
C04352=1031.913,100.142,-98.475,168.895,43.408,158.139
C04353=1031.908,99.893,-98.456,168.892,43.410,158.139
C04354=1031.901,99.644,-98.437,168.889,43.411,158.139
C04355=1031.895,99.395,-98.417,168.888,43.413,158.139
C04356=1031.889,99.146,-98.398,168.885,43.414,158.139
C04357=1031.883,98.896,-98.379,168.882,43.416,158.139
C04358=1031.876,98.646,-98.360,168.881,43.417,158.139
C04359=1031.870,98.398,-98.340,168.878,43.419,158.139
C04360=1031.864,98.149,-98.322,168.875,43.420,158.139
C04361=1031.858,97.899,-98.302,168.873,43.422,158.140
C04362=1031.852,97.650,-98.284,168.871,43.423,158.140
C04363=1031.846,97.401,-98.264,168.868,43.425,158.140
C04364=1031.839,97.152,-98.245,168.866,43.426,158.140
C04365=1031.833,96.903,-98.226,168.864,43.427,158.140
C04366=1031.827,96.653,-98.207,168.862,43.429,158.140
C04367=1031.821,96.404,-98.188,168.859,43.430,158.140
C04368=1031.815,96.155,-98.169,168.857,43.432,158.140
C04369=1031.808,95.906,-98.150,168.855,43.433,158.140
C04370=1031.803,95.657,-98.131,168.852,43.435,158.141
C04371=1031.796,95.407,-98.112,168.849,43.436,158.141
C04372=1031.790,95.158,-98.092,168.848,43.438,158.141
C04373=1031.783,94.909,-98.074,168.845,43.439,158.141
C04374=1031.778,94.659,-98.054,168.842,43.441,158.141
C04375=1031.771,94.410,-98.036,168.840,43.442,158.141
C04376=1031.765,94.162,-98.016,168.838,43.444,158.141
C04377=1031.759,93.912,-97.997,168.836,43.445,158.141
C04378=1031.753,93.663,-97.979,168.833,43.447,158.141
C04379=1031.747,93.414,-97.959,168.830,43.448,158.141
C04380=1031.740,93.164,-97.941,168.829,43.450,158.141
C04381=1031.735,92.915,-97.921,168.826,43.451,158.141
C04382=1031.728,92.630,-97.899,168.823,43.453,158.142
C04383=1031.721,92.345,-97.879,168.821,43.454,158.142
C04384=1031.713,92.059,-97.856,168.818,43.456,158.142
C04385=1031.707,91.773,-97.835,168.815,43.457,158.142
C04386=1031.701,91.524,-97.816,168.812,43.459,158.142
C04387=1031.695,91.275,-97.797,168.811,43.460,158.142
C04388=1031.689,91.025,-97.778,168.808,43.462,158.142
C04389=1031.682,90.776,-97.759,168.806,43.463,158.142
C04390=1031.676,90.527,-97.741,168.804,43.464,158.142
C04391=1031.670,90.278,-97.722,168.801,43.466,158.142
C04392=1031.664,90.029,-97.703,168.799,43.467,158.142
C04393=1031.658,89.779,-97.684,168.797,43.469,158.143
C04394=1031.652,89.530,-97.665,168.795,43.470,158.143
C04395=1031.645,89.281,-97.646,168.792,43.472,158.143
C04396=1031.639,89.032,-97.628,168.789,43.474,158.143
C04397=1031.632,88.783,-97.609,168.788,43.475,158.143
C04398=1031.627,88.534,-97.591,168.785,43.477,158.143
C04399=1031.621,88.285,-97.572,168.782,43.478,158.143
C04400=1031.615,88.036,-97.553,168.781,43.480,158.143
C04401=1031.608,87.786,-97.535,168.778,43.481,158.143
C04402=1031.602,87.537,-97.516,168.775,43.483,158.143
C04403=1031.596,87.288,-97.498,168.774,43.484,158.144
C04404=1031.589,87.039,-97.479,168.771,43.486,158.144
C04405=1031.583,86.789,-97.460,168.768,43.487,158.144
C04406=1031.577,86.540,-97.441,168.766,43.489,158.144
C04407=1031.571,86.290,-97.423,168.764,43.490,158.144
C04408=1031.564,86.041,-97.405,168.762,43.492,158.144
C04409=1031.558,85.792,-97.386,168.759,43.493,158.144
C04410=1031.552,85.543,-97.367,168.757,43.495,158.144
C04411=1031.545,85.294,-97.349,168.755,43.496,158.144
C04412=1031.539,85.044,-97.331,168.752,43.498,158.145
C04413=1031.534,84.795,-97.312,168.750,43.500,158.145
C04414=1031.528,84.546,-97.293,168.748,43.501,158.145
C04415=1031.521,84.297,-97.274,168.745,43.503,158.145
C04416=1031.515,84.047,-97.257,168.742,43.504,158.145
C04417=1031.509,83.798,-97.238,168.741,43.505,158.145
C04418=1031.502,83.549,-97.219,168.738,43.507,158.145
C04419=1031.496,83.300,-97.201,168.736,43.508,158.145
C04420=1031.490,83.050,-97.182,168.734,43.510,158.145
C04421=1031.485,82.802,-97.164,168.731,43.511,158.145
C04422=1031.478,82.552,-97.145,168.729,43.513,158.146
C04423=1031.472,82.303,-97.127,168.726,43.514,158.146
C04424=1031.466,82.054,-97.109,168.725,43.516,158.146
C04425=1031.459,81.804,-97.090,168.722,43.517,158.146
C04426=1031.453,81.555,-97.071,168.719,43.519,158.146
C04427=1031.447,81.306,-97.053,168.717,43.520,158.146
C04428=1031.441,81.057,-97.035,168.715,43.522,158.146
C04429=1031.435,80.808,-97.016,168.712,43.523,158.146
C04430=1031.429,80.558,-96.998,168.710,43.525,158.146
C04431=1031.423,80.309,-96.979,168.708,43.526,158.146
C04432=1031.416,80.059,-96.961,168.706,43.528,158.146
C04433=1031.411,79.811,-96.943,168.703,43.529,158.146
C04434=1031.404,79.562,-96.924,168.700,43.531,158.147
C04435=1031.398,79.312,-96.906,168.699,43.532,158.147
C04436=1031.392,79.063,-96.888,168.696,43.534,158.147
C04437=1031.385,78.814,-96.869,168.694,43.535,158.147
C04438=1031.380,78.564,-96.851,168.692,43.536,158.147
C04439=1031.374,78.315,-96.832,168.689,43.538,158.147
C04440=1031.368,78.065,-96.814,168.687,43.539,158.147
C04441=1031.361,77.816,-96.796,168.685,43.541,158.147
C04442=1031.355,77.566,-96.778,168.683,43.542,158.147
C04443=1031.349,77.318,-96.759,168.680,43.544,158.147
C04444=1031.343,77.068,-96.742,168.677,43.545,158.147
C04445=1031.337,76.819,-96.723,168.676,43.547,158.148
C04446=1031.330,76.534,-96.702,168.673,43.549,158.148
C04447=1031.322,76.249,-96.682,168.670,43.551,158.148
C04448=1031.315,75.963,-96.661,168.668,43.552,158.148
C04449=1031.308,75.677,-96.641,168.665,43.554,158.148
C04450=1031.302,75.428,-96.622,168.662,43.556,158.148
C04451=1031.296,75.179,-96.604,168.659,43.557,158.148
C04452=1031.289,74.929,-96.586,168.658,43.559,158.148
C04453=1031.284,74.680,-96.568,168.655,43.560,158.149
C04454=1031.278,74.431,-96.550,168.653,43.561,158.149
C04455=1031.271,74.181,-96.532,168.651,43.563,158.149
C04456=1031.264,73.932,-96.514,168.648,43.565,158.149
C04457=1031.258,73.684,-96.496,168.646,43.566,158.149
C04458=1031.252,73.434,-96.478,168.644,43.568,158.149
C04459=1031.246,73.184,-96.460,168.641,43.569,158.149
C04460=1031.240,72.935,-96.441,168.639,43.571,158.149
C04461=1031.234,72.686,-96.424,168.637,43.573,158.149
C04462=1031.227,72.437,-96.407,168.635,43.574,158.149
C04463=1031.221,72.187,-96.388,168.632,43.576,158.150
C04464=1031.215,71.938,-96.370,168.629,43.577,158.150
C04465=1031.209,71.689,-96.352,168.628,43.579,158.150
C04466=1031.203,71.440,-96.334,168.625,43.580,158.150
C04467=1031.196,71.190,-96.316,168.622,43.582,158.150
C04468=1031.191,70.941,-96.299,168.621,43.583,158.150
C04469=1031.184,70.692,-96.280,168.618,43.585,158.150
C04470=1031.178,70.442,-96.262,168.616,43.586,158.150
C04471=1031.172,70.193,-96.245,168.614,43.587,158.150
C04472=1031.165,69.944,-96.227,168.611,43.589,158.150
C04473=1031.159,69.695,-96.209,168.609,43.591,158.151
C04474=1031.154,69.446,-96.191,168.606,43.592,158.151
C04475=1031.148,69.196,-96.173,168.604,43.594,158.151
C04476=1031.141,68.947,-96.155,168.602,43.595,158.151
C04477=1031.134,68.697,-96.137,168.599,43.597,158.151
C04478=1031.129,68.448,-96.120,168.598,43.599,158.151
C04479=1031.122,68.199,-96.102,168.595,43.600,158.151
C04480=1031.116,67.949,-96.084,168.592,43.602,158.151
C04481=1031.110,67.700,-96.067,168.591,43.603,158.151
C04482=1031.103,67.451,-96.049,168.588,43.605,158.151
C04483=1031.097,67.201,-96.031,168.585,43.606,158.152
C04484=1031.091,66.952,-96.013,168.583,43.607,158.152
C04485=1031.085,66.703,-95.996,168.581,43.609,158.152
C04486=1031.078,66.453,-95.978,168.579,43.611,158.152
C04487=1031.073,66.204,-95.960,168.576,43.612,158.152
C04488=1031.066,65.955,-95.943,168.574,43.614,158.152
C04489=1031.060,65.706,-95.925,168.572,43.616,158.152
C04490=1031.053,65.457,-95.907,168.569,43.617,158.152
C04491=1031.047,65.207,-95.890,168.567,43.619,158.152
C04492=1031.042,64.958,-95.872,168.565,43.620,158.152
C04493=1031.035,64.709,-95.855,168.562,43.622,158.153
C04494=1031.029,64.459,-95.837,168.560,43.624,158.153
C04495=1031.023,64.210,-95.820,168.558,43.625,158.153
C04496=1031.016,63.961,-95.802,168.555,43.627,158.153
C04497=1031.011,63.711,-95.784,168.554,43.628,158.153
C04498=1031.004,63.462,-95.767,168.551,43.629,158.153
C04499=1030.997,63.213,-95.750,168.548,43.631,158.153
C04500=1030.992,62.964,-95.732,168.547,43.633,158.153
C04501=1030.985,62.714,-95.715,168.544,43.635,158.153
C04502=1030.978,62.465,-95.697,168.541,43.636,158.153
C04503=1030.972,62.216,-95.680,168.539,43.638,158.154
C04504=1030.966,61.966,-95.662,168.537,43.640,158.154
C04505=1030.959,61.718,-95.645,168.534,43.642,158.154
C04506=1030.953,61.467,-95.628,168.531,43.643,158.154
C04507=1030.947,61.218,-95.611,168.530,43.644,158.154
C04508=1030.940,60.969,-95.594,168.527,43.646,158.154
C04509=1030.934,60.719,-95.576,168.525,43.648,158.154
C04510=1030.927,60.434,-95.557,168.522,43.650,158.155
C04511=1030.920,60.148,-95.537,168.519,43.652,158.155
C04512=1030.912,59.863,-95.517,168.517,43.654,158.155
C04513=1030.905,59.577,-95.497,168.514,43.656,158.155
C04514=1030.899,59.327,-95.480,168.511,43.657,158.155
C04515=1030.893,59.078,-95.462,168.510,43.659,158.155
C04516=1030.886,58.829,-95.445,168.507,43.660,158.155
C04517=1030.879,58.580,-95.428,168.504,43.662,158.155
C04518=1030.873,58.330,-95.411,168.503,43.663,158.155
C04519=1030.867,58.081,-95.393,168.500,43.665,158.156
C04520=1030.861,57.831,-95.377,168.497,43.667,158.156
C04521=1030.854,57.582,-95.360,168.496,43.668,158.156
C04522=1030.848,57.333,-95.342,168.493,43.670,158.156
C04523=1030.842,57.084,-95.325,168.490,43.672,158.156
C04524=1030.835,56.834,-95.307,168.489,43.674,158.156
C04525=1030.829,56.585,-95.291,168.486,43.675,158.156
C04526=1030.823,56.335,-95.273,168.483,43.677,158.156
C04527=1030.817,56.087,-95.256,168.482,43.678,158.157
C04528=1030.810,55.837,-95.239,168.479,43.680,158.157
C04529=1030.805,55.587,-95.222,168.476,43.681,158.157
C04530=1030.798,55.338,-95.205,168.475,43.683,158.157
C04531=1030.791,55.089,-95.188,168.472,43.685,158.157
C04532=1030.785,54.839,-95.171,168.469,43.686,158.157
C04533=1030.779,54.590,-95.154,168.468,43.688,158.157
C04534=1030.773,54.341,-95.136,168.465,43.690,158.157
C04535=1030.766,54.092,-95.119,168.462,43.691,158.157
C04536=1030.760,53.842,-95.102,168.461,43.693,158.157
C04537=1030.754,53.593,-95.085,168.458,43.695,158.158
C04538=1030.747,53.344,-95.068,168.455,43.696,158.158
C04539=1030.741,53.094,-95.051,168.453,43.697,158.158
C04540=1030.735,52.844,-95.034,168.451,43.699,158.158
C04541=1030.729,52.596,-95.017,168.448,43.701,158.158
C04542=1030.723,52.346,-95.000,168.446,43.702,158.158
C04543=1030.716,52.097,-94.983,168.444,43.704,158.158
C04544=1030.711,51.848,-94.965,168.442,43.705,158.158
C04545=1030.704,51.598,-94.949,168.439,43.707,158.158
C04546=1030.698,51.349,-94.932,168.437,43.708,158.158
C04547=1030.691,51.099,-94.915,168.435,43.710,158.159
C04548=1030.686,50.850,-94.898,168.432,43.712,158.159
C04549=1030.680,50.601,-94.881,168.429,43.713,158.159
C04550=1030.673,50.351,-94.864,168.428,43.715,158.159
C04551=1030.667,50.103,-94.847,168.425,43.717,158.159
C04552=1030.661,49.852,-94.830,168.422,43.718,158.159
C04553=1030.655,49.603,-94.813,168.421,43.720,158.159
C04554=1030.648,49.355,-94.796,168.418,43.721,158.159
C04555=1030.642,49.105,-94.779,168.415,43.723,158.159
C04556=1030.636,48.856,-94.762,168.414,43.724,158.160
C04557=1030.630,48.606,-94.745,168.411,43.726,158.159
C04558=1030.624,48.357,-94.728,168.409,43.727,158.160
C04559=1030.618,48.107,-94.712,168.407,43.728,158.160
C04560=1030.611,47.858,-94.694,168.404,43.730,158.160
C04561=1030.606,47.608,-94.678,168.402,43.732,158.160
C04562=1030.599,47.360,-94.661,168.399,43.733,158.160
C04563=1030.593,47.110,-94.644,168.397,43.735,158.160
C04564=1030.587,46.861,-94.626,168.395,43.736,158.160
C04565=1030.581,46.611,-94.610,168.392,43.738,158.160
C04566=1030.574,46.362,-94.593,168.390,43.740,158.160
C04567=1030.568,46.112,-94.577,168.388,43.741,158.160
C04568=1030.563,45.863,-94.559,168.385,43.743,158.161
C04569=1030.556,45.613,-94.542,168.384,43.744,158.161
C04570=1030.550,45.365,-94.525,168.381,43.746,158.161
C04571=1030.544,45.115,-94.509,168.378,43.747,158.161
C04572=1030.538,44.866,-94.491,168.376,43.749,158.161
C04573=1030.532,44.616,-94.475,168.374,43.750,158.161
C04574=1030.524,44.331,-94.456,168.371,43.752,158.161
C04575=1030.518,44.045,-94.437,168.368,43.754,158.161
C04576=1030.511,43.759,-94.417,168.366,43.756,158.161
C04577=1030.504,43.473,-94.398,168.363,43.757,158.161
C04578=1030.498,43.223,-94.382,168.360,43.759,158.161
C04579=1030.492,42.973,-94.364,168.359,43.760,158.162
C04580=1030.486,42.724,-94.348,168.356,43.762,158.162
C04581=1030.480,42.475,-94.331,168.353,43.763,158.162
C04582=1030.473,42.225,-94.314,168.352,43.765,158.162
C04583=1030.467,41.976,-94.298,168.349,43.766,158.162
C04584=1030.461,41.727,-94.282,168.346,43.768,158.162
C04585=1030.454,41.477,-94.266,168.345,43.770,158.162
C04586=1030.448,41.228,-94.249,168.342,43.771,158.162
C04587=1030.442,40.979,-94.232,168.339,43.773,158.162
C04588=1030.436,40.729,-94.216,168.338,43.775,158.163
C04589=1030.429,40.479,-94.200,168.335,43.776,158.163
C04590=1030.423,40.231,-94.183,168.332,43.778,158.163
C04591=1030.417,39.981,-94.166,168.331,43.780,158.163
C04592=1030.411,39.732,-94.150,168.328,43.781,158.163
C04593=1030.405,39.482,-94.133,168.325,43.783,158.163
C04594=1030.398,39.233,-94.116,168.324,43.784,158.163
C04595=1030.392,38.984,-94.100,168.321,43.786,158.163
C04596=1030.386,38.735,-94.084,168.318,43.787,158.163
C04597=1030.380,38.484,-94.067,168.316,43.789,158.163
C04598=1030.374,38.235,-94.051,168.314,43.790,158.163
C04599=1030.368,37.986,-94.034,168.311,43.792,158.164
C04600=1030.362,37.737,-94.018,168.308,43.794,158.164
C04601=1030.355,37.487,-94.001,168.307,43.795,158.164
C04602=1030.349,37.238,-93.985,168.304,43.797,158.164
C04603=1030.342,36.989,-93.969,168.301,43.799,158.164
C04604=1030.337,36.739,-93.953,168.300,43.800,158.164
C04605=1030.330,36.489,-93.936,168.297,43.802,158.164
C04606=1030.324,36.240,-93.920,168.294,43.804,158.164
C04607=1030.317,35.991,-93.904,168.293,43.805,158.164
C04608=1030.311,35.741,-93.888,168.290,43.807,158.164
C04609=1030.305,35.492,-93.872,168.287,43.809,158.165
C04610=1030.299,35.242,-93.855,168.285,43.810,158.165
C04611=1030.292,34.993,-93.840,168.283,43.812,158.165
C04612=1030.286,34.744,-93.823,168.280,43.813,158.165
C04613=1030.280,34.494,-93.807,168.278,43.815,158.165
C04614=1030.274,34.245,-93.791,168.276,43.817,158.165
C04615=1030.267,33.995,-93.775,168.273,43.819,158.165
C04616=1030.261,33.746,-93.759,168.271,43.820,158.165
C04617=1030.255,33.497,-93.742,168.268,43.822,158.165
C04618=1030.248,33.248,-93.727,168.266,43.824,158.166
C04619=1030.243,32.998,-93.710,168.263,43.825,158.166
C04620=1030.236,32.748,-93.694,168.261,43.827,158.166
C04621=1030.229,32.499,-93.678,168.259,43.829,158.166
C04622=1030.223,32.250,-93.662,168.257,43.830,158.166
C04623=1030.217,32.000,-93.646,168.254,43.832,158.166
C04624=1030.211,31.751,-93.630,168.251,43.834,158.166
C04625=1030.205,31.502,-93.614,168.250,43.835,158.166
C04626=1030.199,31.253,-93.597,168.247,43.836,158.166
C04627=1030.192,31.003,-93.581,168.244,43.838,158.166
C04628=1030.186,30.754,-93.565,168.243,43.840,158.167
C04629=1030.180,30.504,-93.549,168.240,43.841,158.167
C04630=1030.174,30.255,-93.533,168.237,43.843,158.167
C04631=1030.167,30.005,-93.518,168.234,43.845,158.167
C04632=1030.161,29.756,-93.501,168.233,43.847,158.167
C04633=1030.155,29.507,-93.485,168.230,43.848,158.167
C04634=1030.149,29.257,-93.470,168.227,43.850,158.167
C04635=1030.143,29.008,-93.453,168.226,43.852,158.167
C04636=1030.136,28.758,-93.437,168.223,43.853,158.167
C04637=1030.129,28.509,-93.421,168.220,43.855,158.167
C04638=1030.123,28.223,-93.403,168.218,43.857,158.168
C04639=1030.116,27.937,-93.385,168.215,43.859,158.168
C04640=1030.109,27.651,-93.367,168.213,43.860,158.168
C04641=1030.101,27.365,-93.348,168.210,43.862,158.168
C04642=1030.095,27.115,-93.333,168.207,43.864,158.168
C04643=1030.089,26.866,-93.317,168.204,43.865,158.168
C04644=1030.082,26.617,-93.301,168.202,43.867,158.168
C04645=1030.076,26.367,-93.285,168.200,43.869,158.168
C04646=1030.070,26.118,-93.270,168.197,43.870,158.168
C04647=1030.064,25.868,-93.254,168.195,43.872,158.169
C04648=1030.057,25.619,-93.238,168.192,43.874,158.169
C04649=1030.051,25.369,-93.222,168.191,43.876,158.169
C04650=1030.044,25.120,-93.206,168.188,43.878,158.169
C04651=1030.038,24.870,-93.190,168.185,43.879,158.169
C04652=1030.032,24.621,-93.175,168.183,43.881,158.169
C04653=1030.026,24.371,-93.159,168.181,43.883,158.169
C04654=1030.019,24.122,-93.143,168.178,43.884,158.169
C04655=1030.014,23.872,-93.128,168.175,43.886,158.169
C04656=1030.007,23.623,-93.112,168.173,43.888,158.169
C04657=1030.000,23.374,-93.096,168.171,43.889,158.170
C04658=1029.995,23.124,-93.081,168.169,43.891,158.170
C04659=1029.988,22.875,-93.065,168.166,43.892,158.170
C04660=1029.982,22.625,-93.050,168.163,43.894,158.170
C04661=1029.976,22.376,-93.034,168.162,43.896,158.170
C04662=1029.970,22.127,-93.018,168.159,43.897,158.170
C04663=1029.963,21.877,-93.003,168.156,43.899,158.170
C04664=1029.957,21.628,-92.986,168.154,43.901,158.170
C04665=1029.951,21.378,-92.972,168.152,43.903,158.171
C04666=1029.944,21.129,-92.956,168.149,43.904,158.170
C04667=1029.939,20.879,-92.940,168.147,43.906,158.171
C04668=1029.932,20.630,-92.925,168.144,43.908,158.171
C04669=1029.926,20.381,-92.908,168.142,43.909,158.171
C04670=1029.920,20.131,-92.893,168.139,43.911,158.171
C04671=1029.914,19.882,-92.877,168.137,43.913,158.171
C04672=1029.907,19.632,-92.862,168.134,43.914,158.171
C04673=1029.901,19.383,-92.847,168.132,43.916,158.171
C04674=1029.895,19.133,-92.831,168.130,43.917,158.171
C04675=1029.889,18.884,-92.816,168.127,43.919,158.171
C04676=1029.882,18.635,-92.800,168.125,43.921,158.172
C04677=1029.876,18.385,-92.785,168.122,43.922,158.172
C04678=1029.870,18.136,-92.769,168.120,43.924,158.172
C04679=1029.863,17.886,-92.754,168.118,43.926,158.172
C04680=1029.857,17.637,-92.739,168.115,43.928,158.172
C04681=1029.852,17.388,-92.723,168.112,43.930,158.172
C04682=1029.845,17.138,-92.709,168.110,43.931,158.172
C04683=1029.838,16.889,-92.693,168.108,43.933,158.172
C04684=1029.833,16.639,-92.677,168.105,43.935,158.172
C04685=1029.826,16.390,-92.662,168.103,43.937,158.173
C04686=1029.820,16.140,-92.647,168.100,43.938,158.173
C04687=1029.813,15.891,-92.632,168.098,43.940,158.173
C04688=1029.807,15.641,-92.616,168.096,43.941,158.173
C04689=1029.801,15.392,-92.601,168.093,43.943,158.173
C04690=1029.795,15.142,-92.586,168.090,43.945,158.173
C04691=1029.789,14.893,-92.569,168.088,43.947,158.173
C04692=1029.783,14.644,-92.555,168.086,43.948,158.173
C04693=1029.777,14.394,-92.540,168.083,43.949,158.173
C04694=1029.770,14.145,-92.524,168.080,43.951,158.173
C04695=1029.764,13.895,-92.509,168.078,43.953,158.173
C04696=1029.758,13.645,-92.494,168.076,43.955,158.174
C04697=1029.751,13.396,-92.479,168.073,43.956,158.174
C04698=1029.745,13.147,-92.463,168.071,43.958,158.174
C04699=1029.738,12.897,-92.448,168.068,43.960,158.174
C04700=1029.732,12.647,-92.433,168.066,43.962,158.174
C04701=1029.726,12.398,-92.418,168.063,43.964,158.174
C04702=1029.719,12.113,-92.401,168.060,43.966,158.174
C04703=1029.711,11.829,-92.384,168.058,43.968,158.174
C04704=1029.704,11.544,-92.367,168.055,43.970,158.174
C04705=1029.697,11.259,-92.349,168.052,43.972,158.175
C04706=1029.690,11.010,-92.334,168.050,43.973,158.175
C04707=1029.684,10.760,-92.319,168.047,43.975,158.175
C04708=1029.678,10.511,-92.305,168.045,43.977,158.175
C04709=1029.672,10.261,-92.290,168.042,43.979,158.175
C04710=1029.665,10.012,-92.275,168.039,43.981,158.175
C04711=1029.659,9.762,-92.260,168.037,43.983,158.175
C04712=1029.652,9.512,-92.245,168.034,43.984,158.175
C04713=1029.646,9.263,-92.229,168.032,43.986,158.176
C04714=1029.640,9.014,-92.215,168.030,43.988,158.176
C04715=1029.634,8.765,-92.200,168.027,43.990,158.176
C04716=1029.627,8.515,-92.185,168.025,43.992,158.176
C04717=1029.621,8.265,-92.170,168.022,43.993,158.176
C04718=1029.614,8.016,-92.155,168.019,43.995,158.176
C04719=1029.609,7.767,-92.140,168.018,43.996,158.176
C04720=1029.602,7.517,-92.125,168.015,43.998,158.176
C04721=1029.596,7.267,-92.110,168.012,44.000,158.176
C04722=1029.590,7.018,-92.096,168.010,44.002,158.177
C04723=1029.583,6.768,-92.081,168.007,44.003,158.176
C04724=1029.577,6.519,-92.066,168.004,44.005,158.177
C04725=1029.571,6.269,-92.051,168.003,44.007,158.177
C04726=1029.565,6.020,-92.036,168.000,44.009,158.177
C04727=1029.558,5.770,-92.021,167.997,44.011,158.177
C04728=1029.552,5.521,-92.007,167.995,44.012,158.177
C04729=1029.546,5.272,-91.992,167.992,44.014,158.177
C04730=1029.540,5.022,-91.977,167.989,44.016,158.177
C04731=1029.533,4.772,-91.962,167.987,44.018,158.177
C04732=1029.527,4.523,-91.947,167.985,44.020,158.178
C04733=1029.521,4.274,-91.932,167.982,44.021,158.178
C04734=1029.515,4.024,-91.917,167.980,44.023,158.178
C04735=1029.509,3.775,-91.903,167.977,44.025,158.178
C04736=1029.503,3.525,-91.888,167.974,44.026,158.178
C04737=1029.496,3.276,-91.873,167.972,44.028,158.178
C04738=1029.490,3.026,-91.858,167.970,44.029,158.178
C04739=1029.483,2.777,-91.844,167.967,44.031,158.178
C04740=1029.477,2.527,-91.830,167.965,44.033,158.178
C04741=1029.471,2.277,-91.815,167.962,44.035,158.178
C04742=1029.465,2.028,-91.800,167.959,44.036,158.178
C04743=1029.459,1.779,-91.785,167.957,44.038,158.179
C04744=1029.452,1.529,-91.770,167.955,44.040,158.179
C04745=1029.446,1.280,-91.756,167.952,44.041,158.179
C04746=1029.440,1.031,-91.741,167.950,44.043,158.179
C04747=1029.434,0.781,-91.726,167.947,44.045,158.179
C04748=1029.428,0.531,-91.712,167.945,44.047,158.179
C04749=1029.422,0.282,-91.697,167.942,44.048,158.179
C04750=1029.415,0.032,-91.682,167.940,44.050,158.179
C04751=1029.410,-0.217,-91.667,167.937,44.052,158.179
C04752=1029.403,-0.467,-91.652,167.935,44.053,158.179
C04753=1029.398,-0.716,-91.638,167.932,44.055,158.179
C04754=1029.391,-0.966,-91.624,167.929,44.057,158.180
C04755=1029.385,-1.215,-91.609,167.927,44.059,158.180
C04756=1029.379,-1.464,-91.594,167.924,44.060,158.180
C04757=1029.373,-1.714,-91.579,167.922,44.062,158.180
C04758=1029.367,-1.964,-91.565,167.920,44.064,158.180
C04759=1029.360,-2.213,-91.551,167.917,44.065,158.180
C04760=1029.354,-2.463,-91.536,167.914,44.067,158.180
C04761=1029.348,-2.712,-91.521,167.912,44.069,158.180
C04762=1029.342,-2.962,-91.507,167.909,44.070,158.180
C04763=1029.336,-3.211,-91.493,167.907,44.072,158.180
C04764=1029.330,-3.461,-91.478,167.905,44.074,158.180
C04765=1029.324,-3.710,-91.463,167.902,44.075,158.180
C04766=1029.317,-3.993,-91.447,167.899,44.077,158.181
C04767=1029.310,-4.276,-91.430,167.896,44.080,158.181
C04768=1029.302,-4.558,-91.414,167.893,44.082,158.181
C04769=1029.295,-4.842,-91.398,167.891,44.083,158.181
C04770=1029.289,-5.091,-91.385,167.888,44.085,158.181
C04771=1029.283,-5.341,-91.370,167.885,44.087,158.181
C04772=1029.277,-5.590,-91.355,167.883,44.089,158.181
C04773=1029.270,-5.840,-91.342,167.880,44.090,158.181
C04774=1029.264,-6.089,-91.327,167.877,44.092,158.181
C04775=1029.258,-6.338,-91.313,167.875,44.094,158.182
C04776=1029.251,-6.588,-91.298,167.872,44.096,158.182
C04777=1029.246,-6.838,-91.284,167.869,44.098,158.182
C04778=1029.239,-7.087,-91.270,167.867,44.100,158.182
C04779=1029.233,-7.337,-91.256,167.864,44.102,158.182
C04780=1029.226,-7.586,-91.242,167.861,44.103,158.182
C04781=1029.221,-7.836,-91.228,167.860,44.105,158.182
C04782=1029.214,-8.085,-91.213,167.857,44.107,158.182
C04783=1029.207,-8.335,-91.199,167.855,44.109,158.182
C04784=1029.202,-8.584,-91.185,167.852,44.111,158.183
C04785=1029.195,-8.834,-91.171,167.849,44.113,158.183
C04786=1029.189,-9.083,-91.157,167.847,44.115,158.183
C04787=1029.182,-9.333,-91.143,167.844,44.116,158.183
C04788=1029.176,-9.582,-91.128,167.841,44.118,158.183
C04789=1029.170,-9.832,-91.114,167.839,44.120,158.183
C04790=1029.164,-10.082,-91.101,167.836,44.122,158.183
C04791=1029.158,-10.331,-91.086,167.833,44.123,158.183
C04792=1029.151,-10.580,-91.073,167.831,44.125,158.183
C04793=1029.145,-10.830,-91.058,167.828,44.127,158.183
C04794=1029.139,-11.079,-91.045,167.825,44.129,158.183
C04795=1029.133,-11.329,-91.031,167.824,44.130,158.184
C04796=1029.127,-11.579,-91.016,167.821,44.132,158.184
C04797=1029.121,-11.828,-91.002,167.819,44.134,158.184
C04798=1029.115,-12.078,-90.988,167.816,44.135,158.184
C04799=1029.108,-12.327,-90.974,167.813,44.137,158.184
C04800=1029.102,-12.577,-90.960,167.811,44.139,158.184
C04801=1029.096,-12.826,-90.946,167.808,44.141,158.184
C04802=1029.089,-13.076,-90.932,167.805,44.143,158.184
C04803=1029.083,-13.325,-90.919,167.802,44.144,158.184
C04804=1029.078,-13.575,-90.905,167.800,44.146,158.184
C04805=1029.071,-13.824,-90.890,167.797,44.148,158.184
C04806=1029.065,-14.074,-90.876,167.795,44.150,158.185
C04807=1029.059,-14.324,-90.862,167.792,44.152,158.185
C04808=1029.053,-14.573,-90.848,167.789,44.153,158.185
C04809=1029.047,-14.822,-90.834,167.788,44.155,158.185
C04810=1029.040,-15.072,-90.821,167.785,44.157,158.185
C04811=1029.035,-15.322,-90.807,167.782,44.159,158.185
C04812=1029.028,-15.571,-90.793,167.780,44.160,158.185
C04813=1029.022,-15.821,-90.779,167.777,44.162,158.185
C04814=1029.015,-16.071,-90.765,167.774,44.164,158.185
C04815=1029.009,-16.320,-90.752,167.772,44.166,158.185
C04816=1029.004,-16.569,-90.738,167.769,44.168,158.185
C04817=1028.997,-16.819,-90.724,167.767,44.170,158.186
C04818=1028.990,-17.068,-90.710,167.764,44.172,158.186
C04819=1028.984,-17.318,-90.696,167.761,44.174,158.186
C04820=1028.978,-17.568,-90.683,167.759,44.175,158.186
C04821=1028.972,-17.817,-90.669,167.756,44.177,158.186
C04822=1028.965,-18.067,-90.656,167.753,44.179,158.186
C04823=1028.960,-18.316,-90.642,167.751,44.181,158.186
C04824=1028.953,-18.566,-90.629,167.748,44.183,158.186
C04825=1028.947,-18.816,-90.615,167.745,44.184,158.186
C04826=1028.941,-19.065,-90.601,167.743,44.186,158.187
C04827=1028.935,-19.314,-90.588,167.740,44.188,158.187
C04828=1028.928,-19.564,-90.574,167.738,44.190,158.187
C04829=1028.922,-19.813,-90.560,167.735,44.192,158.187
C04830=1028.915,-20.095,-90.545,167.731,44.194,158.187
C04831=1028.908,-20.376,-90.530,167.729,44.196,158.187
C04832=1028.901,-20.658,-90.515,167.726,44.198,158.187
C04833=1028.894,-20.938,-90.499,167.722,44.200,158.187
C04834=1028.888,-21.188,-90.486,167.720,44.202,158.187
C04835=1028.882,-21.437,-90.472,167.717,44.204,158.187
C04836=1028.875,-21.687,-90.459,167.715,44.206,158.188
C04837=1028.869,-21.937,-90.445,167.712,44.208,158.188
C04838=1028.864,-22.186,-90.431,167.709,44.210,158.188
C04839=1028.857,-22.436,-90.418,167.707,44.212,158.188
C04840=1028.850,-22.685,-90.405,167.704,44.213,158.188
C04841=1028.845,-22.935,-90.391,167.701,44.215,158.188
C04842=1028.839,-23.184,-90.377,167.699,44.217,158.188
C04843=1028.832,-23.434,-90.364,167.696,44.219,158.188
C04844=1028.826,-23.683,-90.351,167.694,44.221,158.188
C04845=1028.820,-23.933,-90.337,167.691,44.223,158.188
C04846=1028.814,-24.182,-90.323,167.688,44.224,158.188
C04847=1028.808,-24.433,-90.310,167.685,44.226,158.189
C04848=1028.801,-24.682,-90.297,167.683,44.228,158.189
C04849=1028.796,-24.932,-90.283,167.680,44.230,158.189
C04850=1028.790,-25.181,-90.270,167.678,44.232,158.189
C04851=1028.783,-25.430,-90.257,167.675,44.234,158.189
C04852=1028.777,-25.680,-90.243,167.672,44.235,158.189
C04853=1028.771,-25.930,-90.229,167.670,44.237,158.189
C04854=1028.765,-26.179,-90.216,167.667,44.239,158.189
C04855=1028.759,-26.429,-90.203,167.664,44.241,158.189
C04856=1028.753,-26.678,-90.190,167.662,44.243,158.189
C04857=1028.747,-26.928,-90.176,167.659,44.245,158.189
C04858=1028.741,-27.178,-90.163,167.656,44.246,158.189
C04859=1028.734,-27.427,-90.149,167.654,44.248,158.190
C04860=1028.728,-27.677,-90.137,167.651,44.250,158.190
C04861=1028.722,-27.926,-90.124,167.648,44.252,158.190
C04862=1028.715,-28.176,-90.110,167.646,44.254,158.190
C04863=1028.709,-28.425,-90.097,167.643,44.255,158.190
C04864=1028.703,-28.675,-90.084,167.641,44.257,158.190
C04865=1028.697,-28.924,-90.071,167.638,44.259,158.190
C04866=1028.691,-29.174,-90.058,167.635,44.261,158.190
C04867=1028.684,-29.424,-90.045,167.633,44.263,158.190
C04868=1028.678,-29.674,-90.031,167.630,44.265,158.191
C04869=1028.672,-29.923,-90.018,167.628,44.267,158.191
C04870=1028.666,-30.173,-90.006,167.624,44.269,158.191
C04871=1028.660,-30.422,-89.992,167.621,44.271,158.191
C04872=1028.654,-30.672,-89.980,167.619,44.273,158.191
C04873=1028.648,-30.921,-89.967,167.616,44.275,158.191
C04874=1028.641,-31.171,-89.953,167.614,44.277,158.191
C04875=1028.635,-31.421,-89.940,167.611,44.279,158.191
C04876=1028.629,-31.670,-89.927,167.608,44.281,158.191
C04877=1028.623,-31.920,-89.914,167.606,44.283,158.192
C04878=1028.617,-32.169,-89.901,167.603,44.285,158.192
C04879=1028.610,-32.419,-89.888,167.600,44.286,158.192
C04880=1028.604,-32.669,-89.875,167.598,44.288,158.192
C04881=1028.598,-32.918,-89.863,167.595,44.290,158.192
C04882=1028.592,-33.167,-89.850,167.592,44.292,158.192
C04883=1028.585,-33.417,-89.837,167.590,44.294,158.192
C04884=1028.579,-33.667,-89.824,167.586,44.296,158.192
C04885=1028.573,-33.917,-89.811,167.584,44.298,158.192
C04886=1028.566,-34.166,-89.797,167.581,44.300,158.192
C04887=1028.561,-34.416,-89.785,167.578,44.302,158.192
C04888=1028.554,-34.665,-89.772,167.576,44.304,158.193
C04889=1028.548,-34.915,-89.759,167.573,44.305,158.193
C04890=1028.542,-35.164,-89.746,167.571,44.307,158.193
C04891=1028.536,-35.414,-89.733,167.568,44.309,158.193
C04892=1028.530,-35.663,-89.720,167.565,44.311,158.193
C04893=1028.522,-36.011,-89.702,167.562,44.313,158.193
C04894=1028.514,-36.350,-89.686,167.557,44.316,158.193
C04895=1028.507,-36.590,-89.673,167.554,44.318,158.193
C04896=1028.501,-36.831,-89.660,167.552,44.320,158.193
C04897=1028.496,-37.071,-89.648,167.550,44.321,158.193
C04898=1028.490,-37.312,-89.636,167.548,44.323,158.194
C04899=1028.484,-37.552,-89.623,167.545,44.325,158.194
C04900=1028.479,-37.792,-89.611,167.542,44.327,158.194
C04901=1028.472,-38.033,-89.598,167.540,44.328,158.194
C04902=1028.466,-38.283,-89.586,167.537,44.330,158.194
C04903=1028.460,-38.533,-89.573,167.534,44.332,158.194
C04904=1028.454,-38.782,-89.560,167.531,44.334,158.194
C04905=1028.448,-39.032,-89.547,167.528,44.336,158.194
C04906=1028.442,-39.281,-89.535,167.526,44.338,158.194
C04907=1028.435,-39.531,-89.522,167.523,44.340,158.194
C04908=1028.430,-39.781,-89.509,167.520,44.342,158.194
C04909=1028.423,-40.030,-89.497,167.518,44.344,158.195
C04910=1028.417,-40.280,-89.485,167.515,44.346,158.195
C04911=1028.411,-40.529,-89.472,167.511,44.348,158.195
C04912=1028.405,-40.778,-89.460,167.509,44.350,158.195
C04913=1028.399,-41.028,-89.447,167.506,44.352,158.195
C04914=1028.393,-41.278,-89.435,167.504,44.354,158.195
C04915=1028.386,-41.527,-89.422,167.501,44.356,158.195
C04916=1028.380,-41.777,-89.410,167.498,44.358,158.195
C04917=1028.374,-42.027,-89.397,167.496,44.360,158.195
C04918=1028.368,-42.276,-89.385,167.492,44.362,158.195
C04919=1028.362,-42.526,-89.373,167.490,44.364,158.195
C04920=1028.355,-42.775,-89.359,167.487,44.366,158.196
C04921=1028.349,-43.025,-89.347,167.484,44.368,158.196
C04922=1028.343,-43.275,-89.335,167.482,44.370,158.196
C04923=1028.337,-43.525,-89.322,167.479,44.372,158.196
C04924=1028.330,-43.774,-89.310,167.477,44.374,158.196
C04925=1028.325,-44.023,-89.298,167.473,44.376,158.196
C04926=1028.319,-44.273,-89.286,167.470,44.378,158.196
C04927=1028.312,-44.522,-89.273,167.468,44.380,158.196
C04928=1028.306,-44.772,-89.260,167.465,44.382,158.196
C04929=1028.300,-45.022,-89.248,167.462,44.384,158.196
C04930=1028.294,-45.272,-89.236,167.460,44.386,158.197
C04931=1028.288,-45.522,-89.223,167.457,44.388,158.197
C04932=1028.282,-45.771,-89.211,167.454,44.390,158.197
C04933=1028.276,-46.020,-89.199,167.451,44.392,158.197
C04934=1028.270,-46.270,-89.187,167.448,44.394,158.197
C04935=1028.264,-46.520,-89.174,167.446,44.396,158.197
C04936=1028.257,-46.770,-89.162,167.443,44.397,158.197
C04937=1028.251,-47.020,-89.150,167.441,44.399,158.197
C04938=1028.246,-47.269,-89.137,167.438,44.401,158.197
C04939=1028.239,-47.518,-89.125,167.434,44.403,158.197
C04940=1028.234,-47.768,-89.113,167.432,44.405,158.198
C04941=1028.227,-48.018,-89.101,167.429,44.407,158.198
C04942=1028.221,-48.268,-89.088,167.427,44.409,158.198
C04943=1028.216,-48.517,-89.076,167.424,44.411,158.198
C04944=1028.209,-48.766,-89.064,167.421,44.413,158.198
C04945=1028.203,-49.016,-89.052,167.418,44.415,158.198
C04946=1028.197,-49.266,-89.039,167.415,44.417,158.198
C04947=1028.191,-49.515,-89.027,167.412,44.419,158.198
C04948=1028.185,-49.765,-89.015,167.410,44.421,158.198
C04949=1028.179,-50.015,-89.002,167.407,44.422,158.198
C04950=1028.173,-50.264,-88.990,167.404,44.424,158.198
C04951=1028.167,-50.514,-88.978,167.402,44.426,158.199
C04952=1028.161,-50.763,-88.966,167.398,44.429,158.199
C04953=1028.155,-51.013,-88.954,167.396,44.431,158.199
C04954=1028.149,-51.263,-88.942,167.393,44.433,158.199
C04955=1028.142,-51.513,-88.930,167.391,44.435,158.199
C04956=1028.136,-51.762,-88.919,167.387,44.437,158.199
C04957=1028.130,-52.011,-88.906,167.384,44.439,158.199
C04958=1028.123,-52.293,-88.894,167.381,44.442,158.199
C04959=1028.116,-52.573,-88.880,167.378,44.444,158.199
C04960=1028.109,-52.854,-88.867,167.375,44.447,158.200
C04961=1028.101,-53.135,-88.853,167.371,44.449,158.200
C04962=1028.096,-53.385,-88.841,167.369,44.451,158.200
C04963=1028.090,-53.634,-88.830,167.366,44.454,158.200
C04964=1028.083,-53.884,-88.818,167.364,44.455,158.200
C04965=1028.077,-54.134,-88.807,167.360,44.458,158.200
C04966=1028.071,-54.384,-88.794,167.358,44.460,158.200
C04967=1028.065,-54.633,-88.783,167.355,44.462,158.200
C04968=1028.058,-54.883,-88.771,167.353,44.464,158.201
C04969=1028.052,-55.132,-88.759,167.349,44.466,158.201
C04970=1028.046,-55.381,-88.747,167.346,44.468,158.201
C04971=1028.040,-55.632,-88.736,167.344,44.470,158.201
C04972=1028.033,-55.881,-88.724,167.341,44.472,158.201
C04973=1028.027,-56.130,-88.712,167.337,44.474,158.201
C04974=1028.021,-56.380,-88.701,167.335,44.477,158.201
C04975=1028.015,-56.630,-88.689,167.332,44.479,158.201
C04976=1028.009,-56.880,-88.678,167.330,44.481,158.201
C04977=1028.003,-57.129,-88.666,167.326,44.483,158.202
C04978=1027.996,-57.379,-88.654,167.324,44.485,158.202
C04979=1027.991,-57.629,-88.642,167.321,44.487,158.202
C04980=1027.984,-57.878,-88.630,167.318,44.489,158.202
C04981=1027.978,-58.128,-88.619,167.315,44.492,158.202
C04982=1027.972,-58.377,-88.607,167.312,44.494,158.202
C04983=1027.966,-58.628,-88.596,167.310,44.496,158.202
C04984=1027.960,-58.877,-88.584,167.307,44.498,158.202
C04985=1027.954,-59.127,-88.573,167.304,44.500,158.202
C04986=1027.947,-59.376,-88.561,167.301,44.502,158.202
C04987=1027.941,-59.625,-88.549,167.298,44.504,158.203
C04988=1027.936,-59.876,-88.537,167.296,44.506,158.203
C04989=1027.930,-60.125,-88.527,167.292,44.508,158.203
C04990=1027.923,-60.375,-88.515,167.290,44.510,158.203
C04991=1027.918,-60.624,-88.504,167.287,44.512,158.203
C04992=1027.911,-60.874,-88.492,167.285,44.514,158.203
C04993=1027.905,-61.124,-88.480,167.281,44.516,158.203
C04994=1027.899,-61.373,-88.468,167.278,44.518,158.203
C04995=1027.893,-61.623,-88.457,167.276,44.521,158.204
C04996=1027.887,-61.872,-88.445,167.272,44.523,158.204
C04997=1027.881,-62.123,-88.434,167.270,44.525,158.204
C04998=1027.875,-62.372,-88.422,167.267,44.527,158.204
C04999=1027.869,-62.622,-88.411,167.264,44.529,158.204
C05000=1027.863,-62.871,-88.400,167.261,44.531,158.204
C05001=1027.857,-63.121,-88.388,167.258,44.533,158.204
C05002=1027.851,-63.370,-88.377,167.256,44.535,158.204
C05003=1027.845,-63.620,-88.365,167.253,44.537,158.204
C05004=1027.839,-63.870,-88.354,167.250,44.540,158.204
C05005=1027.833,-64.120,-88.342,167.247,44.542,158.205
C05006=1027.827,-64.369,-88.331,167.244,44.544,158.205
C05007=1027.821,-64.619,-88.320,167.242,44.546,158.205
C05008=1027.816,-64.869,-88.308,167.238,44.548,158.205
C05009=1027.809,-65.118,-88.296,167.236,44.550,158.205
C05010=1027.803,-65.368,-88.285,167.233,44.552,158.205
C05011=1027.797,-65.618,-88.274,167.230,44.554,158.205
C05012=1027.791,-65.867,-88.262,167.227,44.556,158.205
C05013=1027.785,-66.116,-88.252,167.224,44.558,158.205
C05014=1027.779,-66.367,-88.240,167.222,44.561,158.205
C05015=1027.774,-66.616,-88.229,167.219,44.563,158.206
C05016=1027.767,-66.866,-88.217,167.216,44.565,158.206
C05017=1027.761,-67.116,-88.206,167.213,44.567,158.206
C05018=1027.755,-67.366,-88.195,167.210,44.569,158.206
C05019=1027.749,-67.615,-88.183,167.207,44.571,158.206
C05020=1027.744,-67.864,-88.172,167.204,44.573,158.206
C05021=1027.738,-68.115,-88.160,167.201,44.575,158.206
C05022=1027.731,-68.396,-88.148,167.198,44.577,158.206
C05023=1027.725,-68.678,-88.136,167.195,44.580,158.206
C05024=1027.717,-68.960,-88.122,167.192,44.582,158.206
///RCONF 1,0,0,1,0,0,0,0,0,0,0,0,0,0,0,0,0,0,0,0,0,0,0,0
C05025=1027.711,-69.242,-88.110,167.188,44.585,158.206
C05026=1027.704,-69.492,-88.099,167.186,44.587,158.207
C05027=1027.699,-69.742,-88.087,167.183,44.589,158.207
C05028=1027.694,-69.991,-88.076,167.180,44.591,158.207
C05029=1027.687,-70.241,-88.064,167.177,44.593,158.207
C05030=1027.681,-70.490,-88.054,167.174,44.595,158.207
C05031=1027.675,-70.740,-88.043,167.172,44.597,158.207
C05032=1027.669,-70.990,-88.031,167.168,44.599,158.207
C05033=1027.663,-71.240,-88.021,167.166,44.601,158.207
C05034=1027.658,-71.489,-88.009,167.163,44.603,158.207
C05035=1027.652,-71.740,-87.998,167.160,44.605,158.207
C05036=1027.646,-71.988,-87.986,167.157,44.607,158.207
C05037=1027.640,-72.238,-87.975,167.154,44.609,158.207
C05038=1027.634,-72.487,-87.965,167.152,44.611,158.208
C05039=1027.628,-72.738,-87.953,167.149,44.613,158.208
C05040=1027.622,-72.987,-87.942,167.145,44.615,158.208
C05041=1027.617,-73.237,-87.931,167.143,44.617,158.208
C05042=1027.611,-73.487,-87.920,167.140,44.620,158.208
C05043=1027.605,-73.737,-87.909,167.137,44.622,158.208
C05044=1027.600,-73.986,-87.898,167.134,44.624,158.208
C05045=1027.594,-74.236,-87.887,167.132,44.626,158.208
C05046=1027.587,-74.486,-87.876,167.129,44.628,158.208
C05047=1027.582,-74.735,-87.865,167.125,44.630,158.208
C05048=1027.576,-74.985,-87.854,167.123,44.632,158.208
C05049=1027.569,-75.235,-87.843,167.120,44.634,158.209
C05050=1027.563,-75.485,-87.833,167.117,44.637,158.209
C05051=1027.558,-75.734,-87.822,167.114,44.639,158.209
C05052=1027.552,-75.984,-87.812,167.111,44.641,158.209
C05053=1027.546,-76.234,-87.800,167.108,44.643,158.209
C05054=1027.540,-76.483,-87.789,167.105,44.645,158.209
C05055=1027.534,-76.733,-87.779,167.103,44.647,158.209
C05056=1027.528,-76.982,-87.768,167.099,44.650,158.209
C05057=1027.522,-77.232,-87.757,167.097,44.651,158.209
C05058=1027.516,-77.482,-87.747,167.093,44.654,158.210
C05059=1027.510,-77.732,-87.736,167.091,44.656,158.210
C05060=1027.504,-77.981,-87.725,167.088,44.658,158.210
C05061=1027.499,-78.231,-87.714,167.084,44.660,158.210
C05062=1027.492,-78.481,-87.704,167.082,44.663,158.210
C05063=1027.486,-78.731,-87.693,167.079,44.665,158.210
C05064=1027.480,-78.980,-87.683,167.076,44.667,158.210
C05065=1027.475,-79.230,-87.672,167.073,44.669,158.210
C05066=1027.469,-79.479,-87.661,167.071,44.671,158.210
C05067=1027.464,-79.729,-87.651,167.067,44.674,158.211
C05068=1027.456,-79.979,-87.640,167.065,44.676,158.211
C05069=1027.451,-80.229,-87.629,167.062,44.678,158.211
C05070=1027.445,-80.479,-87.619,167.059,44.681,158.211
C05071=1027.439,-80.728,-87.609,167.056,44.683,158.211
C05072=1027.433,-80.978,-87.598,167.052,44.685,158.211
C05073=1027.426,-81.228,-87.588,167.050,44.688,158.211
C05074=1027.421,-81.478,-87.577,167.047,44.690,158.211
C05075=1027.414,-81.727,-87.567,167.044,44.693,158.212
C05076=1027.409,-81.977,-87.556,167.041,44.695,158.212
C05077=1027.403,-82.226,-87.546,167.038,44.697,158.212
C05078=1027.397,-82.476,-87.536,167.035,44.699,158.212
C05079=1027.391,-82.726,-87.525,167.033,44.701,158.212
C05080=1027.384,-82.976,-87.515,167.029,44.704,158.212
C05081=1027.378,-83.226,-87.504,167.027,44.706,158.212
C05082=1027.372,-83.475,-87.494,167.023,44.708,158.212
C05083=1027.367,-83.725,-87.484,167.021,44.711,158.213
C05084=1027.361,-83.974,-87.473,167.018,44.713,158.213
C05085=1027.355,-84.224,-87.463,167.015,44.715,158.213
C05086=1027.348,-84.509,-87.452,167.011,44.718,158.213
C05087=1027.341,-84.792,-87.440,167.008,44.721,158.213
C05088=1027.334,-85.076,-87.428,167.004,44.724,158.213
C05089=1027.327,-85.361,-87.416,167.002,44.726,158.213
C05090=1027.321,-85.611,-87.406,166.998,44.729,158.213
C05091=1027.315,-85.860,-87.396,166.996,44.731,158.214
C05092=1027.309,-86.110,-87.386,166.992,44.733,158.214
C05093=1027.303,-86.360,-87.375,166.990,44.735,158.214
C05094=1027.297,-86.609,-87.366,166.987,44.737,158.214
C05095=1027.292,-86.859,-87.355,166.984,44.740,158.214
C05096=1027.286,-87.109,-87.344,166.981,44.742,158.214
C05097=1027.280,-87.358,-87.334,166.978,44.744,158.214
C05098=1027.274,-87.608,-87.324,166.975,44.747,158.214
C05099=1027.268,-87.858,-87.314,166.973,44.749,158.215
C05100=1027.262,-88.108,-87.304,166.969,44.751,158.215
C05101=1027.256,-88.357,-87.294,166.967,44.754,158.215
C05102=1027.250,-88.607,-87.283,166.963,44.756,158.215
C05103=1027.244,-88.857,-87.274,166.960,44.758,158.215
C05104=1027.239,-89.107,-87.263,166.957,44.761,158.215
C05105=1027.232,-89.356,-87.253,166.954,44.763,158.215
C05106=1027.227,-89.606,-87.243,166.952,44.765,158.215
C05107=1027.221,-89.856,-87.233,166.948,44.768,158.215
C05108=1027.215,-90.105,-87.223,166.946,44.770,158.216
C05109=1027.209,-90.355,-87.213,166.942,44.772,158.216
C05110=1027.203,-90.605,-87.203,166.940,44.775,158.216
C05111=1027.197,-90.854,-87.193,166.937,44.777,158.216
C05112=1027.192,-91.104,-87.183,166.934,44.779,158.216
C05113=1027.186,-91.354,-87.173,166.931,44.782,158.216
C05114=1027.180,-91.603,-87.162,166.928,44.784,158.216
C05115=1027.174,-91.853,-87.153,166.925,44.786,158.216
C05116=1027.169,-92.103,-87.143,166.923,44.788,158.216
C05117=1027.162,-92.353,-87.133,166.919,44.791,158.217
C05118=1027.157,-92.602,-87.122,166.916,44.793,158.217
C05119=1027.150,-92.852,-87.113,166.913,44.795,158.217
C05120=1027.145,-93.102,-87.102,166.910,44.797,158.217
C05121=1027.139,-93.352,-87.093,166.908,44.799,158.217
C05122=1027.134,-93.602,-87.083,166.904,44.802,158.217
C05123=1027.128,-93.851,-87.073,166.902,44.804,158.217
C05124=1027.122,-94.101,-87.063,166.898,44.806,158.217
C05125=1027.116,-94.351,-87.053,166.896,44.809,158.217
C05126=1027.111,-94.601,-87.043,166.893,44.811,158.218
C05127=1027.104,-94.851,-87.033,166.890,44.813,158.218
C05128=1027.099,-95.099,-87.023,166.887,44.816,158.218
C05129=1027.093,-95.349,-87.013,166.884,44.818,158.218
C05130=1027.088,-95.599,-87.003,166.881,44.820,158.218
C05131=1027.081,-95.849,-86.993,166.879,44.823,158.218
C05132=1027.076,-96.099,-86.983,166.875,44.825,158.218
C05133=1027.070,-96.349,-86.974,166.872,44.827,158.218
C05134=1027.065,-96.598,-86.964,166.869,44.830,158.218
C05135=1027.059,-96.848,-86.954,166.866,44.832,158.219
C05136=1027.053,-97.098,-86.943,166.864,44.834,158.219
C05137=1027.047,-97.347,-86.934,166.860,44.837,158.219
C05138=1027.041,-97.598,-86.924,166.858,44.839,158.219
C05139=1027.036,-97.847,-86.915,166.854,44.842,158.219
C05140=1027.030,-98.096,-86.905,166.852,44.844,158.219
C05141=1027.024,-98.346,-86.895,166.848,44.846,158.219
C05142=1027.017,-98.596,-86.886,166.846,44.848,158.219
C05143=1027.013,-98.845,-86.876,166.842,44.851,158.220
C05144=1027.006,-99.095,-86.867,166.840,44.853,158.220
C05145=1027.001,-99.346,-86.858,166.836,44.856,158.220
C05146=1026.994,-99.595,-86.848,166.834,44.858,158.220
C05147=1026.989,-99.846,-86.838,166.830,44.861,158.220
C05148=1026.983,-100.095,-86.829,166.828,44.863,158.220
C05149=1026.977,-100.344,-86.819,166.826,44.866,158.220
C05150=1026.970,-100.631,-86.808,166.822,44.868,158.220
C05151=1026.963,-100.917,-86.797,166.819,44.871,158.221
C05152=1026.957,-101.203,-86.786,166.815,44.874,158.221
C05153=1026.951,-101.490,-86.775,166.812,44.877,158.221
C05154=1026.944,-101.739,-86.766,166.808,44.879,158.221
C05155=1026.938,-101.989,-86.756,166.806,44.882,158.221
C05156=1026.933,-102.239,-86.748,166.802,44.884,158.221
C05157=1026.928,-102.489,-86.738,166.800,44.886,158.221
C05158=1026.921,-102.739,-86.728,166.796,44.889,158.221
C05159=1026.916,-102.988,-86.719,166.794,44.891,158.222
C05160=1026.910,-103.238,-86.709,166.790,44.893,158.222
C05161=1026.903,-103.487,-86.700,166.788,44.896,158.222
C05162=1026.898,-103.737,-86.691,166.784,44.898,158.222
C05163=1026.893,-103.987,-86.681,166.782,44.901,158.222
C05164=1026.887,-104.237,-86.671,166.778,44.903,158.222
C05165=1026.881,-104.486,-86.662,166.776,44.906,158.222
C05166=1026.875,-104.737,-86.653,166.773,44.908,158.222
C05167=1026.869,-104.986,-86.644,166.770,44.911,158.223
C05168=1026.863,-105.235,-86.635,166.767,44.913,158.223
C05169=1026.858,-105.486,-86.624,166.764,44.916,158.223
C05170=1026.852,-105.736,-86.616,166.761,44.918,158.223
C05171=1026.847,-105.985,-86.606,166.758,44.921,158.223
C05172=1026.840,-106.235,-86.597,166.755,44.923,158.223
C05173=1026.835,-106.485,-86.588,166.752,44.926,158.223
C05174=1026.829,-106.734,-86.579,166.749,44.928,158.224
C05175=1026.823,-106.984,-86.569,166.746,44.930,158.224
C05176=1026.818,-107.234,-86.561,166.744,44.933,158.224
C05177=1026.811,-107.484,-86.551,166.740,44.935,158.224
C05178=1026.806,-107.733,-86.542,166.738,44.938,158.224
C05179=1026.800,-107.983,-86.533,166.734,44.940,158.224
C05180=1026.794,-108.233,-86.524,166.732,44.943,158.224
C05181=1026.788,-108.483,-86.515,166.728,44.946,158.224
C05182=1026.782,-108.733,-86.505,166.726,44.948,158.225
C05183=1026.777,-108.982,-86.497,166.722,44.951,158.225
C05184=1026.771,-109.232,-86.487,166.720,44.953,158.225
C05185=1026.765,-109.481,-86.478,166.716,44.956,158.225
///RCONF 1,0,0,0,0,0,0,0,0,0,0,0,0,0,0,0,0,0,0,0,0,0,0,0
C05186=1026.759,-109.732,-86.469,166.714,44.958,158.225
C05187=1026.754,-109.981,-86.460,166.710,44.960,158.225
C05188=1026.748,-110.231,-86.451,166.708,44.963,158.225
C05189=1026.742,-110.481,-86.442,166.704,44.965,158.225
C05190=1026.737,-110.731,-86.433,166.702,44.968,158.226
C05191=1026.730,-110.980,-86.424,166.698,44.971,158.226
C05192=1026.725,-111.230,-86.415,166.696,44.973,158.226
C05193=1026.719,-111.480,-86.406,166.692,44.976,158.226
C05194=1026.714,-111.730,-86.397,166.690,44.978,158.226
C05195=1026.708,-111.980,-86.388,166.686,44.981,158.226
C05196=1026.702,-112.229,-86.379,166.684,44.983,158.227
C05197=1026.696,-112.480,-86.370,166.681,44.986,158.227
C05198=1026.691,-112.729,-86.361,166.678,44.988,158.227
C05199=1026.685,-112.979,-86.352,166.675,44.991,158.227
C05200=1026.679,-113.228,-86.343,166.672,44.993,158.227
C05201=1026.674,-113.478,-86.335,166.669,44.996,158.227
C05202=1026.668,-113.728,-86.326,166.666,44.998,158.227
C05203=1026.663,-113.977,-86.316,166.663,45.001,158.227
C05204=1026.657,-114.228,-86.308,166.660,45.003,158.227
C05205=1026.651,-114.477,-86.300,166.657,45.006,158.228
C05206=1026.645,-114.727,-86.290,166.654,45.009,158.228
C05207=1026.639,-114.977,-86.282,166.651,45.011,158.228
C05208=1026.634,-115.227,-86.273,166.647,45.014,158.228
C05209=1026.628,-115.476,-86.264,166.645,45.017,158.228
C05210=1026.623,-115.726,-86.255,166.641,45.019,158.228
C05211=1026.616,-115.976,-86.247,166.639,45.021,158.228
C05212=1026.611,-116.225,-86.238,166.636,45.024,158.229
C05213=1026.605,-116.476,-86.229,166.633,45.026,158.229
C05214=1026.598,-116.761,-86.219,166.630,45.029,158.229
C05215=1026.592,-117.048,-86.209,166.626,45.032,158.229
C05216=1026.585,-117.333,-86.199,166.623,45.036,158.229
C05217=1026.579,-117.619,-86.189,166.620,45.039,158.229
C05218=1026.573,-117.869,-86.181,166.616,45.041,158.230
C05219=1026.567,-118.119,-86.172,166.614,45.044,158.230
C05220=1026.562,-118.369,-86.164,166.610,45.047,158.230
C05221=1026.556,-118.618,-86.154,166.608,45.049,158.230
C05222=1026.550,-118.868,-86.146,166.604,45.051,158.230
C05223=1026.544,-119.118,-86.138,166.601,45.054,158.230
C05224=1026.539,-119.367,-86.129,166.599,45.057,158.230
C05225=1026.533,-119.618,-86.120,166.595,45.059,158.230
C05226=1026.527,-119.867,-86.112,166.593,45.062,158.231
C05227=1026.522,-120.117,-86.104,166.589,45.065,158.231
C05228=1026.516,-120.367,-86.094,166.587,45.067,158.231
C05229=1026.511,-120.616,-86.086,166.583,45.070,158.231
C05230=1026.505,-120.866,-86.078,166.581,45.073,158.231
C05231=1026.499,-121.116,-86.069,166.577,45.075,158.231
C05232=1026.493,-121.366,-86.061,166.575,45.077,158.232
C05233=1026.488,-121.616,-86.052,166.572,45.080,158.232
C05234=1026.482,-121.866,-86.044,166.569,45.083,158.232
C05235=1026.476,-122.115,-86.035,166.566,45.085,158.232
C05236=1026.471,-122.365,-86.027,166.563,45.088,158.232
C05237=1026.466,-122.615,-86.018,166.560,45.091,158.232
C05238=1026.459,-122.865,-86.010,166.556,45.093,158.232
C05239=1026.454,-123.115,-86.002,166.554,45.096,158.233
C05240=1026.449,-123.364,-85.993,166.551,45.099,158.233
C05241=1026.443,-123.614,-85.985,166.548,45.101,158.233
C05242=1026.437,-123.864,-85.976,166.545,45.104,158.233
C05243=1026.432,-124.114,-85.968,166.542,45.106,158.233
C05244=1026.426,-124.363,-85.960,166.539,45.109,158.233
C05245=1026.420,-124.613,-85.952,166.537,45.112,158.234
C05246=1026.414,-124.863,-85.943,166.533,45.114,158.234
C05247=1026.408,-125.113,-85.935,166.531,45.117,158.234
C05248=1026.403,-125.363,-85.926,166.527,45.120,158.234
C05249=1026.397,-125.612,-85.918,166.524,45.123,158.234
C05250=1026.392,-125.862,-85.910,166.521,45.126,158.234
C05251=1026.385,-126.112,-85.902,166.518,45.128,158.234
C05252=1026.380,-126.362,-85.894,166.515,45.130,158.234
C05253=1026.375,-126.612,-85.885,166.512,45.133,158.235
C05254=1026.369,-126.861,-85.878,166.510,45.136,158.235
C05255=1026.364,-127.111,-85.869,166.506,45.139,158.235
C05256=1026.357,-127.361,-85.861,166.503,45.141,158.235
C05257=1026.352,-127.611,-85.852,166.500,45.144,158.235
C05258=1026.346,-127.860,-85.844,166.497,45.147,158.235
C05259=1026.341,-128.109,-85.836,166.494,45.149,158.235
C05260=1026.337,-128.359,-85.827,166.492,45.151,158.236
C05261=1026.332,-128.609,-85.817,166.489,45.152,158.235
C05262=1026.329,-128.859,-85.807,166.486,45.154,158.235
C05263=1026.326,-129.109,-85.797,166.484,45.154,158.235
C05264=1026.322,-129.358,-85.785,166.481,45.154,158.235
C05265=1026.321,-129.608,-85.773,166.478,45.154,158.235
C05266=1026.320,-129.857,-85.761,166.476,45.153,158.234
C05267=1026.319,-130.107,-85.747,166.474,45.151,158.234
C05268=1026.319,-130.357,-85.734,166.472,45.150,158.233
C05269=1026.319,-130.607,-85.719,166.470,45.147,158.233
C05270=1026.320,-130.857,-85.704,166.468,45.144,158.232
C05271=1026.321,-131.107,-85.689,166.466,45.141,158.231
C05272=1026.323,-131.356,-85.673,166.464,45.138,158.231
C05273=1026.326,-131.606,-85.656,166.462,45.133,158.230
C05274=1026.329,-131.857,-85.640,166.461,45.128,158.229
C05275=1026.332,-132.106,-85.622,166.459,45.123,158.228
C05276=1026.337,-132.356,-85.604,166.458,45.117,158.226
C05277=1026.341,-132.606,-85.584,166.456,45.111,158.225
C05278=1026.037,-132.631,-85.908,166.409,45.374,158.264
C05279=1026.031,-132.382,-85.926,166.410,45.380,158.266
C05280=1026.027,-132.132,-85.945,166.411,45.386,158.267
C05281=1026.024,-131.882,-85.963,166.413,45.391,158.268
C05282=1026.021,-131.633,-85.980,166.414,45.396,158.269
C05283=1026.018,-131.383,-85.997,166.416,45.400,158.270
C05284=1026.016,-131.132,-86.013,166.418,45.404,158.270
C05285=1026.015,-130.882,-86.028,166.419,45.407,158.271
C05286=1026.014,-130.632,-86.043,166.422,45.410,158.272
C05287=1026.013,-130.383,-86.057,166.424,45.412,158.272
C05288=1026.013,-130.133,-86.071,166.426,45.414,158.273
C05289=1026.014,-129.884,-86.084,166.428,45.416,158.273
C05290=1026.016,-129.634,-86.097,166.431,45.417,158.274
C05291=1026.018,-129.384,-86.109,166.433,45.417,158.274
C05292=1026.020,-129.134,-86.120,166.435,45.417,158.274
C05293=1026.023,-128.884,-86.131,166.438,45.416,158.275
C05294=1026.026,-128.635,-86.141,166.441,45.415,158.275
C05295=1026.031,-128.385,-86.151,166.444,45.414,158.275
C05296=1026.036,-128.135,-86.160,166.447,45.412,158.275
C05297=1026.041,-127.886,-86.168,166.449,45.409,158.275
C05298=1026.046,-127.636,-86.177,166.452,45.406,158.274
C05299=1026.052,-127.387,-86.185,166.455,45.404,158.274
C05300=1026.058,-127.137,-86.193,166.458,45.401,158.274
C05301=1026.064,-126.888,-86.201,166.462,45.398,158.274
C05302=1026.069,-126.637,-86.209,166.464,45.396,158.274
C05303=1026.075,-126.388,-86.217,166.467,45.393,158.274
C05304=1026.080,-126.137,-86.226,166.470,45.390,158.273
C05305=1026.086,-125.888,-86.234,166.473,45.388,158.273
C05306=1026.092,-125.638,-86.242,166.477,45.385,158.273
C05307=1026.097,-125.389,-86.251,166.479,45.382,158.273
C05308=1026.103,-125.139,-86.258,166.482,45.379,158.273
C05309=1026.109,-124.888,-86.267,166.485,45.376,158.273
C05310=1026.115,-124.639,-86.274,166.488,45.373,158.273
C05311=1026.120,-124.389,-86.283,166.491,45.370,158.272
C05312=1026.125,-124.139,-86.291,166.494,45.368,158.272
C05313=1026.132,-123.889,-86.300,166.497,45.365,158.272
C05314=1026.137,-123.639,-86.308,166.500,45.363,158.272
C05315=1026.142,-123.390,-86.317,166.503,45.360,158.272
C05316=1026.147,-123.140,-86.325,166.506,45.358,158.272
C05317=1026.154,-122.890,-86.333,166.509,45.355,158.272
C05318=1026.159,-122.640,-86.342,166.512,45.352,158.271
C05319=1026.165,-122.390,-86.350,166.515,45.349,158.271
C05320=1026.171,-122.141,-86.358,166.518,45.346,158.271
C05321=1026.176,-121.891,-86.367,166.521,45.344,158.271
C05322=1026.182,-121.641,-86.376,166.524,45.341,158.271
C05323=1026.187,-121.391,-86.384,166.526,45.339,158.271
C05324=1026.193,-121.142,-86.392,166.530,45.336,158.271
C05325=1026.199,-120.891,-86.401,166.533,45.333,158.270
C05326=1026.204,-120.642,-86.409,166.536,45.331,158.270
C05327=1026.210,-120.393,-86.419,166.539,45.328,158.270
C05328=1026.216,-120.142,-86.427,166.541,45.325,158.270
C05329=1026.222,-119.893,-86.435,166.545,45.323,158.270
C05330=1026.227,-119.643,-86.444,166.547,45.320,158.270
C05331=1026.232,-119.393,-86.452,166.551,45.317,158.270
C05332=1026.239,-119.143,-86.460,166.554,45.314,158.269
C05333=1026.244,-118.894,-86.469,166.557,45.312,158.269
C05334=1026.249,-118.644,-86.477,166.560,45.309,158.269
C05335=1026.255,-118.394,-86.487,166.562,45.306,158.269
C05336=1026.261,-118.145,-86.495,166.566,45.303,158.269
C05337=1026.267,-117.894,-86.504,166.568,45.301,158.269
C05338=1026.273,-117.644,-86.512,166.572,45.299,158.269
C05339=1026.279,-117.359,-86.522,166.575,45.296,158.268
C05340=1026.286,-117.073,-86.533,166.578,45.292,158.268
C05341=1026.292,-116.787,-86.542,166.582,45.289,158.268
C05342=1026.299,-116.501,-86.552,166.585,45.286,158.268
C05343=1026.304,-116.251,-86.560,166.589,45.284,158.268
C05344=1026.310,-116.002,-86.570,166.591,45.281,158.268
C05345=1026.316,-115.752,-86.578,166.594,45.278,158.267
C05346=1026.321,-115.502,-86.587,166.597,45.275,158.267
C05347=1026.327,-115.252,-86.595,166.600,45.273,158.267
C05348=1026.333,-115.003,-86.604,166.604,45.270,158.267
C05349=1026.339,-114.753,-86.613,166.606,45.268,158.267
C05350=1026.344,-114.503,-86.622,166.609,45.265,158.267
C05351=1026.350,-114.253,-86.631,166.612,45.263,158.267
C05352=1026.356,-114.003,-86.640,166.615,45.260,158.266
C05353=1026.361,-113.754,-86.648,166.618,45.257,158.266
C05354=1026.367,-113.504,-86.658,166.621,45.255,158.266
C05355=1026.372,-113.254,-86.666,166.624,45.252,158.266
C05356=1026.378,-113.004,-86.675,166.627,45.249,158.266
C05357=1026.384,-112.755,-86.684,166.630,45.247,158.266
C05358=1026.390,-112.505,-86.692,166.633,45.244,158.266
C05359=1026.396,-112.255,-86.702,166.636,45.241,158.265
C05360=1026.402,-112.005,-86.711,166.639,45.239,158.265
C05361=1026.407,-111.755,-86.719,166.642,45.236,158.265
C05362=1026.413,-111.506,-86.729,166.645,45.234,158.265
C05363=1026.418,-111.256,-86.737,166.648,45.231,158.265
C05364=1026.425,-111.006,-86.747,166.651,45.229,158.265
C05365=1026.430,-110.756,-86.755,166.654,45.226,158.265
C05366=1026.436,-110.507,-86.765,166.657,45.224,158.265
C05367=1026.441,-110.257,-86.773,166.660,45.221,158.264
C05368=1026.448,-110.007,-86.783,166.663,45.219,158.264
C05369=1026.453,-109.757,-86.791,166.666,45.216,158.264
C05370=1026.459,-109.507,-86.801,166.669,45.213,158.264
C05371=1026.464,-109.258,-86.809,166.672,45.211,158.264
C05372=1026.470,-109.008,-86.819,166.675,45.208,158.264
C05373=1026.476,-108.758,-86.827,166.678,45.205,158.264
C05374=1026.482,-108.508,-86.837,166.681,45.203,158.264
C05375=1026.487,-108.259,-86.845,166.684,45.200,158.263
C05376=1026.493,-108.009,-86.855,166.687,45.197,158.263
C05377=1026.499,-107.759,-86.865,166.689,45.195,158.263
C05378=1026.505,-107.509,-86.873,166.693,45.192,158.263
C05379=1026.511,-107.260,-86.883,166.695,45.190,158.263
C05380=1026.516,-107.010,-86.891,166.699,45.187,158.263
C05381=1026.522,-106.760,-86.901,166.701,45.185,158.262
C05382=1026.528,-106.511,-86.910,166.705,45.183,158.262
C05383=1026.534,-106.261,-86.919,166.707,45.180,158.262
C05384=1026.540,-106.011,-86.928,166.711,45.177,158.262
C05385=1026.545,-105.761,-86.938,166.713,45.175,158.262
C05386=1026.551,-105.511,-86.947,166.716,45.172,158.262
C05387=1026.557,-105.261,-86.956,166.719,45.170,158.262
C05388=1026.562,-105.012,-86.966,166.722,45.167,158.262
C05389=1026.569,-104.762,-86.975,166.726,45.165,158.262
C05390=1026.574,-104.513,-86.984,166.728,45.162,158.261
C05391=1026.580,-104.263,-86.993,166.732,45.159,158.261
C05392=1026.585,-104.013,-87.003,166.734,45.157,158.261
C05393=1026.591,-103.763,-87.012,166.738,45.154,158.261
C05394=1026.597,-103.513,-87.021,166.740,45.152,158.261
C05395=1026.603,-103.263,-87.031,166.744,45.149,158.261
C05396=1026.609,-103.014,-87.040,166.746,45.147,158.261
C05397=1026.615,-102.764,-87.050,166.750,45.144,158.260
C05398=1026.620,-102.514,-87.059,166.752,45.142,158.260
C05399=1026.625,-102.265,-87.068,166.756,45.139,158.260
C05400=1026.632,-102.015,-87.078,166.758,45.137,158.260
C05401=1026.638,-101.765,-87.088,166.762,45.135,158.260
C05402=1026.643,-101.516,-87.097,166.764,45.132,158.260
